    // Detect ON/OFF state change
    IF aUnits[i].bPresVal <> aPrevState[i] THEN
        // --------------------------------------------------------
        // (a) Send TwinCAT message as before
        // --------------------------------------------------------
        IF aUnits[i].bPresVal THEN
            sMsgText := CONCAT(stUnit.sUnitName, ' is Turned ON');
        ELSE
            sMsgText := CONCAT(stUnit.sUnitName, ' is Turned OFF');
        END_IF

        fbMsg.CreateEx(TC_EVENTS.UnitPowerStatus.EventPowerStatus, 0);
        fbMsg.ipArguments.AddString(sMsgText);
        fbMsg.Send(0);

        // --------------------------------------------------------
        // (b) Push event to global CSV queue (for P_CSVWrite_TextMode)
        // --------------------------------------------------------
        IF g_iCount < g_CSV_BUF_SIZE THEN
            g_aUnitName[g_iWriteIdx] := stUnit.sUnitName;
            g_aState[g_iWriteIdx]    := aUnits[i].bPresVal;
            g_iWriteIdx := g_iWriteIdx + 1;
            IF g_iWriteIdx > g_CSV_BUF_SIZE THEN g_iWriteIdx := 1; END_IF
            g_iCount := g_iCount + 1;
        END_IF

        // --------------------------------------------------------
        // (c) Update previous state
        // --------------------------------------------------------
        aPrevState[i] := aUnits[i].bPresVal;
    END_IF
END_FOR

// ------------------------------------------------------------
// Optional debug info
// ------------------------------------------------------------
sDebug := CONCAT('Queued=', INT_TO_STRING(g_iCount));

END_FUNCTION_BLOCK

// ---- POUs/FB_EventLogger/FB_EventFMZ2.TcPOU
FUNCTION_BLOCK FB_EventFMZ2
VAR_INPUT
	FB_Bacnet : FB_BACnet_DAIKIN_MasterStation_III_No_1;
END_VAR
VAR_OUTPUT
	sDebug : STRING(200);
END_VAR
VAR
	fbMsg : FB_TcMessage;
	aUnits : ARRAY[1..8] OF AC_Unit_Status;
	stUnit   : AC_Unit_Status;
	i: INT;
	sMsgText: STRING;

END_VAR
VAR RETAIN
	aPrevState : ARRAY[1..8] OF BOOL := [FALSE(*8*)];
END_VAR


aUnits[1].bPresVal := FB_Bacnet.StartStopStatus_096.bPresVal;
aUnits[1].sUnitName := 'FMZ-PC-1 (3-00)';
aUnits[2].bPresVal := FB_Bacnet.StartStopStatus_097.bPresVal;
aUnits[2].sUnitName := 'FMZ-PC-2 (3-01)';
aUnits[3].bPresVal := FB_Bacnet.StartStopStatus_098.bPresVal;
aUnits[3].sUnitName := 'FMZ-PC-3 (3-02)';
aUnits[4].bPresVal := FB_Bacnet.StartStopStatus_099.bPresVal;
aUnits[4].sUnitName := 'FMZ-PC-4 (3-03)';
aUnits[5].bPresVal := FB_Bacnet.StartStopStatus_100.bPresVal;
aUnits[5].sUnitName := 'FMZ-PC-5 (3-04)';
aUnits[6].bPresVal := FB_Bacnet.StartStopStatus_101.bPresVal;
aUnits[6].sUnitName := 'FMZ-PC-6 (3-05)';
aUnits[7].bPresVal := FB_Bacnet.StartStopStatus_102.bPresVal;
aUnits[7].sUnitName := 'FMZ-PC-7 (3-06)';
aUnits[8].bPresVal := FB_Bacnet.StartStopStatus_103.bPresVal;
aUnits[8].sUnitName := 'FMZ-PC-8 (3-07)';

FOR i := 1 TO 8 DO
    stUnit := aUnits[i];

    // Detect ON/OFF state change
    IF aUnits[i].bPresVal <> aPrevState[i] THEN
        // --------------------------------------------------------
        // (a) Send TwinCAT message as before
        // --------------------------------------------------------
        IF aUnits[i].bPresVal THEN
            sMsgText := CONCAT(stUnit.sUnitName, ' is Turned ON');
        ELSE
            sMsgText := CONCAT(stUnit.sUnitName, ' is Turned OFF');
        END_IF

        fbMsg.CreateEx(TC_EVENTS.UnitPowerStatus.EventPowerStatus, 0);
        fbMsg.ipArguments.AddString(sMsgText);
        fbMsg.Send(0);

        // --------------------------------------------------------
        // (b) Push event to global CSV queue (for P_CSVWrite_TextMode)
        // --------------------------------------------------------
        IF g_iCount < g_CSV_BUF_SIZE THEN
            g_aUnitName[g_iWriteIdx] := stUnit.sUnitName;
            g_aState[g_iWriteIdx]    := aUnits[i].bPresVal;
            g_iWriteIdx := g_iWriteIdx + 1;
            IF g_iWriteIdx > g_CSV_BUF_SIZE THEN g_iWriteIdx := 1; END_IF
            g_iCount := g_iCount + 1;
        END_IF

        // --------------------------------------------------------
        // (c) Update previous state
        // --------------------------------------------------------
        aPrevState[i] := aUnits[i].bPresVal;
    END_IF
END_FOR

// ------------------------------------------------------------
// Optional debug info
// ------------------------------------------------------------
sDebug := CONCAT('Queued=', INT_TO_STRING(g_iCount));

END_FUNCTION_BLOCK

// ---- POUs/FB_EventLogger/FB_EventF2.TcPOU
FUNCTION_BLOCK FB_EventF2
VAR_INPUT
	FB_Bacnet : FB_BACnet_DAIKIN_MasterStation_III_No_1;
END_VAR
VAR_OUTPUT
	sDebug : STRING(200);
END_VAR
VAR
	fbMsg : FB_TcMessage;
	aUnits : ARRAY[1..23] OF AC_Unit_Status;
	stUnit   : AC_Unit_Status;
	i: INT;
	sMsgText: STRING;
END_VAR
VAR RETAIN
	aPrevState : ARRAY[1..23] OF BOOL := [FALSE(*23*)];
END_VAR


aUnits[1].bPresVal := FB_Bacnet.StartStopStatus_128.bPresVal;
aUnits[1].sUnitName := 'F2-1 (1-00)';
aUnits[2].bPresVal := FB_Bacnet.StartStopStatus_129.bPresVal;
aUnits[2].sUnitName := 'F2-2 (1-01)';
aUnits[3].bPresVal := FB_Bacnet.StartStopStatus_130.bPresVal;
aUnits[3].sUnitName := 'F2-3 (1-02)';
aUnits[4].bPresVal := FB_Bacnet.StartStopStatus_131.bPresVal;
aUnits[4].sUnitName := 'F2-4 (1-03)';
aUnits[5].bPresVal := FB_Bacnet.StartStopStatus_132.bPresVal;
aUnits[5].sUnitName := 'F2-5 (1-04)';
aUnits[6].bPresVal := FB_Bacnet.StartStopStatus_133.bPresVal;
aUnits[6].sUnitName := 'F2-6 (1-05)';
aUnits[7].bPresVal := FB_Bacnet.StartStopStatus_134.bPresVal;
aUnits[7].sUnitName := 'F2-7 (1-06)';
aUnits[8].bPresVal := FB_Bacnet.StartStopStatus_135.bPresVal;
aUnits[8].sUnitName := 'F2-8 (1-07)';
aUnits[9].bPresVal := FB_Bacnet.StartStopStatus_136.bPresVal;
aUnits[9].sUnitName := 'F2-9 (1-08)';
aUnits[10].bPresVal := FB_Bacnet.StartStopStatus_137.bPresVal;
aUnits[10].sUnitName := 'F2-10 (1-09)';
aUnits[11].bPresVal := FB_Bacnet.StartStopStatus_138.bPresVal;
aUnits[11].sUnitName := 'F2-11 (1-10)';
aUnits[12].bPresVal := FB_Bacnet.StartStopStatus_139.bPresVal;
aUnits[12].sUnitName := 'F2-12 (1-11)';
//aUnits[13].bPresVal := FB_Bacnet.StartStopStatus_140.bPresVal;
//aUnits[13].sUnitName := 'F2-13 (1-12)';
aUnits[14].bPresVal := FB_Bacnet.StartStopStatus_141.bPresVal;
aUnits[14].sUnitName := 'F2-14 (1-13)';
aUnits[15].bPresVal := FB_Bacnet.StartStopStatus_142.bPresVal;
aUnits[15].sUnitName := 'F2-15 (1-14)';
aUnits[16].bPresVal := FB_Bacnet.StartStopStatus_143.bPresVal;
aUnits[16].sUnitName := 'F2-16 (1-15)';
aUnits[17].bPresVal := FB_Bacnet.StartStopStatus_144.bPresVal;
aUnits[17].sUnitName := 'F2-17 (2-00)';
aUnits[18].bPresVal := FB_Bacnet.StartStopStatus_145.bPresVal;
aUnits[18].sUnitName := 'F2-18 (2-01)';
aUnits[19].bPresVal := FB_Bacnet.StartStopStatus_146.bPresVal;
aUnits[19].sUnitName := 'F2-19 (2-02)';
aUnits[20].bPresVal := FB_Bacnet.StartStopStatus_147.bPresVal;
aUnits[20].sUnitName := 'F2-20 (2-03)';
aUnits[21].bPresVal := FB_Bacnet.StartStopStatus_148.bPresVal;
aUnits[21].sUnitName := 'F2-21 (2-04)';
aUnits[22].bPresVal := FB_Bacnet.StartStopStatus_176.bPresVal;
aUnits[22].sUnitName := 'F2-IT-1 (4-00)';
//aUnits[23].bPresVal := FB_Bacnet.StartStopStatus_177.bPresVal;
//aUnits[23].sUnitName := 'F2-IT-2 (4-01)';

FOR i := 1 TO 23 DO
    stUnit := aUnits[i];

    // Detect ON/OFF state change
    IF aUnits[i].bPresVal <> aPrevState[i] THEN
        // --------------------------------------------------------
        // (a) Send TwinCAT message as before
        // --------------------------------------------------------
        IF aUnits[i].bPresVal THEN
            sMsgText := CONCAT(stUnit.sUnitName, ' is Turned ON');
        ELSE
            sMsgText := CONCAT(stUnit.sUnitName, ' is Turned OFF');
        END_IF

        fbMsg.CreateEx(TC_EVENTS.UnitPowerStatus.EventPowerStatus, 0);
        fbMsg.ipArguments.AddString(sMsgText);
        fbMsg.Send(0);

        // --------------------------------------------------------
        // (b) Push event to global CSV queue (for P_CSVWrite_TextMode)
        // --------------------------------------------------------
        IF g_iCount < g_CSV_BUF_SIZE THEN
            g_aUnitName[g_iWriteIdx] := stUnit.sUnitName;
            g_aState[g_iWriteIdx]    := aUnits[i].bPresVal;
            g_iWriteIdx := g_iWriteIdx + 1;
            IF g_iWriteIdx > g_CSV_BUF_SIZE THEN g_iWriteIdx := 1; END_IF
            g_iCount := g_iCount + 1;
        END_IF

        // --------------------------------------------------------
        // (c) Update previous state
        // --------------------------------------------------------
        aPrevState[i] := aUnits[i].bPresVal;
    END_IF
END_FOR

// ------------------------------------------------------------
// Optional debug info
// ------------------------------------------------------------
sDebug := CONCAT('Queued=', INT_TO_STRING(g_iCount));

END_FUNCTION_BLOCK

// ---- POUs/FB_EventLogger/FB_EventF3.TcPOU
FUNCTION_BLOCK FB_EventF3
VAR_INPUT
	FB_Bacnet : FB_BACnet_DAIKIN_MasterStation_III_No_1;
END_VAR
VAR_OUTPUT
	sDebug : STRING(200);
END_VAR
VAR
	fbMsg : FB_TcMessage;
	aUnits : ARRAY[1..22] OF AC_Unit_Status;
	stUnit   : AC_Unit_Status;
	i: INT;
	sMsgText: STRING;

END_VAR
VAR RETAIN
	aPrevState : ARRAY[1..22] OF BOOL := [FALSE(*22*)];
END_VAR


//aUnits[1].bPresVal := FB_Bacnet.StartStopStatus_192.bPresVal;
//aUnits[1].sUnitName := 'F3-1 (1-00)';
aUnits[2].bPresVal := FB_Bacnet.StartStopStatus_193.bPresVal;
aUnits[2].sUnitName := 'F3-2 (1-01)';
aUnits[3].bPresVal := FB_Bacnet.StartStopStatus_194.bPresVal;
aUnits[3].sUnitName := 'F3-3 (1-02)';
aUnits[4].bPresVal := FB_Bacnet.StartStopStatus_195.bPresVal;
aUnits[4].sUnitName := 'F3-4 (1-03)';
aUnits[5].bPresVal := FB_Bacnet.StartStopStatus_196.bPresVal;
aUnits[5].sUnitName := 'F3-5 (1-04)';
aUnits[6].bPresVal := FB_Bacnet.StartStopStatus_197.bPresVal;
aUnits[6].sUnitName := 'F3-6 (1-05)';
aUnits[7].bPresVal := FB_Bacnet.StartStopStatus_198.bPresVal;
aUnits[7].sUnitName := 'F3-7 (1-06)';
aUnits[8].bPresVal := FB_Bacnet.StartStopStatus_199.bPresVal;
aUnits[8].sUnitName := 'F3-8 (1-07)';
aUnits[9].bPresVal := FB_Bacnet.StartStopStatus_200.bPresVal;
aUnits[9].sUnitName := 'F3-9 (1-08)';
aUnits[10].bPresVal := FB_Bacnet.StartStopStatus_201.bPresVal;
aUnits[10].sUnitName := 'F3-10 (1-09)';
aUnits[11].bPresVal := FB_Bacnet.StartStopStatus_202.bPresVal;
aUnits[11].sUnitName := 'F3-11 (1-10)';
aUnits[12].bPresVal := FB_Bacnet.StartStopStatus_203.bPresVal;
aUnits[12].sUnitName := 'F3-12 (1-11)';
aUnits[13].bPresVal := FB_Bacnet.StartStopStatus_204.bPresVal;
aUnits[13].sUnitName := 'F3-13 (1-12)';
aUnits[14].bPresVal := FB_Bacnet.StartStopStatus_205.bPresVal;
aUnits[14].sUnitName := 'F3-14 (1-13)';
aUnits[15].bPresVal := FB_Bacnet.StartStopStatus_206.bPresVal;
aUnits[15].sUnitName := 'F3-15 (1-14)';
aUnits[16].bPresVal := FB_Bacnet.StartStopStatus_207.bPresVal;
aUnits[16].sUnitName := 'F3-16 (1-15)';
aUnits[17].bPresVal := FB_Bacnet.StartStopStatus_208.bPresVal;
aUnits[17].sUnitName := 'F3-17 (2-00)';
aUnits[18].bPresVal := FB_Bacnet.StartStopStatus_209.bPresVal;
aUnits[18].sUnitName := 'F3-18 (2-01)';
aUnits[19].bPresVal := FB_Bacnet.StartStopStatus_210.bPresVal;
aUnits[19].sUnitName := 'F3-19 (2-02)';
aUnits[20].bPresVal := FB_Bacnet.StartStopStatus_211.bPresVal;
aUnits[20].sUnitName := 'F3-20 (2-03)';
aUnits[21].bPresVal := FB_Bacnet.StartStopStatus_212.bPresVal;
aUnits[21].sUnitName := 'F3-21 (2-04)';
aUnits[22].bPresVal := FB_Bacnet.StartStopStatus_224.bPresVal;
aUnits[22].sUnitName := 'F3-Lobi (3-00)';

FOR i := 1 TO 22 DO
    stUnit := aUnits[i];

    // Detect ON/OFF state change
    IF aUnits[i].bPresVal <> aPrevState[i] THEN
        // --------------------------------------------------------
        // (a) Send TwinCAT message as before
        // --------------------------------------------------------
        IF aUnits[i].bPresVal THEN
            sMsgText := CONCAT(stUnit.sUnitName, ' is Turned ON');
        ELSE
            sMsgText := CONCAT(stUnit.sUnitName, ' is Turned OFF');
        END_IF

        fbMsg.CreateEx(TC_EVENTS.UnitPowerStatus.EventPowerStatus, 0);
        fbMsg.ipArguments.AddString(sMsgText);
        fbMsg.Send(0);

        // --------------------------------------------------------
        // (b) Push event to global CSV queue (for P_CSVWrite_TextMode)
        // --------------------------------------------------------
        IF g_iCount < g_CSV_BUF_SIZE THEN
            g_aUnitName[g_iWriteIdx] := stUnit.sUnitName;
            g_aState[g_iWriteIdx]    := aUnits[i].bPresVal;
            g_iWriteIdx := g_iWriteIdx + 1;
            IF g_iWriteIdx > g_CSV_BUF_SIZE THEN g_iWriteIdx := 1; END_IF
            g_iCount := g_iCount + 1;
        END_IF

        // --------------------------------------------------------
        // (c) Update previous state
        // --------------------------------------------------------
        aPrevState[i] := aUnits[i].bPresVal;
    END_IF
END_FOR

// ------------------------------------------------------------
// Optional debug info
// ------------------------------------------------------------
sDebug := CONCAT('Queued=', INT_TO_STRING(g_iCount));

END_FUNCTION_BLOCK

// ---- POUs/FB_EventLogger/FB_EventF5.TcPOU
FUNCTION_BLOCK FB_EventF5
VAR_INPUT
	FB_Bacnet : FB_BACnet_DAIKIN_MasterStation_III_No_2;
    FB_Bacnet_b : FB_BACnet_DAIKIN_MasterStation_III_No_1;
END_VAR
VAR_OUTPUT
	sDebug : STRING(200);
END_VAR
VAR
	fbMsg : FB_TcMessage;
	aUnits : ARRAY[1..22] OF AC_Unit_Status;
	stUnit   : AC_Unit_Status;
	i: INT;
	sMsgText: STRING;

END_VAR
VAR RETAIN
	aPrevState : ARRAY[1..22] OF BOOL := [FALSE(*22*)];
END_VAR


aUnits[1].bPresVal := FB_Bacnet.StartStopStatus_000.bPresVal;
aUnits[1].sUnitName := 'F5-A1 (1-00)';
aUnits[2].bPresVal := FB_Bacnet.StartStopStatus_001.bPresVal;
aUnits[2].sUnitName := 'F5-A2 (1-01)';
aUnits[3].bPresVal := FB_Bacnet.StartStopStatus_002.bPresVal;
aUnits[3].sUnitName := 'F5-A3 (1-02)';
aUnits[4].bPresVal := FB_Bacnet.StartStopStatus_003.bPresVal;
aUnits[4].sUnitName := 'F5-A4 (1-03)';
aUnits[5].bPresVal := FB_Bacnet.StartStopStatus_004.bPresVal;
aUnits[5].sUnitName := 'F5-B1 (1-04)';
aUnits[6].bPresVal := FB_Bacnet.StartStopStatus_005.bPresVal;
aUnits[6].sUnitName := 'F5-B2 (1-05)';
aUnits[7].bPresVal := FB_Bacnet.StartStopStatus_006.bPresVal;
aUnits[7].sUnitName := 'F5-C1 (1-06)';
aUnits[8].bPresVal := FB_Bacnet.StartStopStatus_007.bPresVal;
aUnits[8].sUnitName := 'F5-C2 (1-07)';
aUnits[9].bPresVal := FB_Bacnet.StartStopStatus_008.bPresVal;
aUnits[9].sUnitName := 'F5-D1 (1-08)';
aUnits[10].bPresVal := FB_Bacnet.StartStopStatus_009.bPresVal;
aUnits[10].sUnitName := 'F5-D2 (1-09)';
aUnits[11].bPresVal := FB_Bacnet.StartStopStatus_010.bPresVal;
aUnits[11].sUnitName := 'F5-D3 (1-10)';
aUnits[12].bPresVal := FB_Bacnet.StartStopStatus_011.bPresVal;
aUnits[12].sUnitName := 'F5-D4 (1-11)';
aUnits[13].bPresVal := FB_Bacnet.StartStopStatus_012.bPresVal;
aUnits[13].sUnitName := 'F5-D5 (1-12)';
aUnits[14].bPresVal := FB_Bacnet.StartStopStatus_013.bPresVal;
aUnits[14].sUnitName := 'F5-D6 (1-13)';
aUnits[15].bPresVal := FB_Bacnet.StartStopStatus_014.bPresVal;
aUnits[15].sUnitName := 'F5-E1 (1-14)';
aUnits[16].bPresVal := FB_Bacnet.StartStopStatus_015.bPresVal;
aUnits[16].sUnitName := 'F5-E2 (1-15)';
aUnits[17].bPresVal := FB_Bacnet.StartStopStatus_016.bPresVal;
aUnits[17].sUnitName := 'F5-F1 (2-00)';
aUnits[18].bPresVal := FB_Bacnet.StartStopStatus_017.bPresVal;
aUnits[18].sUnitName := 'F5-F2 (2-01)';
aUnits[19].bPresVal := FB_Bacnet.StartStopStatus_018.bPresVal;
aUnits[19].sUnitName := 'F5-G1 (2-02)';
aUnits[20].bPresVal := FB_Bacnet.StartStopStatus_019.bPresVal;
aUnits[20].sUnitName := 'F5-G2 (2-03)';
aUnits[21].bPresVal := FB_Bacnet.StartStopStatus_020.bPresVal;
aUnits[21].sUnitName := 'F5-G3 (2-04)';
aUnits[22].bPresVal := FB_Bacnet_b.StartStopStatus_225.bPresVal;
aUnits[22].sUnitName := 'F5-Lobi (3-01)';

FOR i := 1 TO 22 DO
    stUnit := aUnits[i];

    // Detect ON/OFF state change
    IF aUnits[i].bPresVal <> aPrevState[i] THEN
        // --------------------------------------------------------
        // (a) Send TwinCAT message as before
        // --------------------------------------------------------
        IF aUnits[i].bPresVal THEN
            sMsgText := CONCAT(stUnit.sUnitName, ' is Turned ON');
        ELSE
            sMsgText := CONCAT(stUnit.sUnitName, ' is Turned OFF');
        END_IF

        fbMsg.CreateEx(TC_EVENTS.UnitPowerStatus.EventPowerStatus, 0);
        fbMsg.ipArguments.AddString(sMsgText);
        fbMsg.Send(0);

        // --------------------------------------------------------
        // (b) Push event to global CSV queue (for P_CSVWrite_TextMode)
        // --------------------------------------------------------
        IF g_iCount < g_CSV_BUF_SIZE THEN
            g_aUnitName[g_iWriteIdx] := stUnit.sUnitName;
            g_aState[g_iWriteIdx]    := aUnits[i].bPresVal;
            g_iWriteIdx := g_iWriteIdx + 1;
            IF g_iWriteIdx > g_CSV_BUF_SIZE THEN g_iWriteIdx := 1; END_IF
            g_iCount := g_iCount + 1;
        END_IF

        // --------------------------------------------------------
        // (c) Update previous state
        // --------------------------------------------------------
        aPrevState[i] := aUnits[i].bPresVal;
    END_IF
END_FOR

// ------------------------------------------------------------
// Optional debug info
// ------------------------------------------------------------
sDebug := CONCAT('Queued=', INT_TO_STRING(g_iCount));

END_FUNCTION_BLOCK

// ---- POUs/FB_EventLogger/FB_EventF6.TcPOU
FUNCTION_BLOCK FB_EventF6
VAR_INPUT
	FB_Bacnet : FB_BACnet_DAIKIN_MasterStation_III_No_2;
    FB_Bacnet_b : FB_BACnet_DAIKIN_MasterStation_III_No_1;
END_VAR
VAR_OUTPUT
	sDebug : STRING(200);
END_VAR
VAR
	fbMsg : FB_TcMessage;
	aUnits : ARRAY[1..22] OF AC_Unit_Status;
	stUnit   : AC_Unit_Status;
	i: INT;
	sMsgText: STRING;

END_VAR
VAR RETAIN
	aPrevState : ARRAY[1..22] OF BOOL := [FALSE(*22*)];
END_VAR


aUnits[1].bPresVal := FB_Bacnet.StartStopStatus_064.bPresVal;
aUnits[1].sUnitName := 'F6-A1 (1-00)';
aUnits[2].bPresVal := FB_Bacnet.StartStopStatus_065.bPresVal;
aUnits[2].sUnitName := 'F6-A2 (1-01)';
aUnits[3].bPresVal := FB_Bacnet.StartStopStatus_066.bPresVal;
aUnits[3].sUnitName := 'F6-A3 (1-02)';
aUnits[4].bPresVal := FB_Bacnet.StartStopStatus_067.bPresVal;
aUnits[4].sUnitName := 'F6-A4 (1-03)';
aUnits[5].bPresVal := FB_Bacnet.StartStopStatus_068.bPresVal;
aUnits[5].sUnitName := 'F6-B1 (1-04)';
aUnits[6].bPresVal := FB_Bacnet.StartStopStatus_069.bPresVal;
aUnits[6].sUnitName := 'F6-B2 (1-05)';
aUnits[7].bPresVal := FB_Bacnet.StartStopStatus_070.bPresVal;
aUnits[7].sUnitName := 'F6-C1 (1-06)';
aUnits[8].bPresVal := FB_Bacnet.StartStopStatus_071.bPresVal;
aUnits[8].sUnitName := 'F6-C2 (1-07)';
aUnits[9].bPresVal := FB_Bacnet.StartStopStatus_072.bPresVal;
aUnits[9].sUnitName := 'F6-D1 (1-08)';
aUnits[10].bPresVal := FB_Bacnet.StartStopStatus_073.bPresVal;
aUnits[10].sUnitName := 'F6-D2 (1-09)';
aUnits[11].bPresVal := FB_Bacnet.StartStopStatus_074.bPresVal;
aUnits[11].sUnitName := 'F6-D3 (1-10)';
aUnits[12].bPresVal := FB_Bacnet.StartStopStatus_075.bPresVal;
aUnits[12].sUnitName := 'F6-D4 (1-11)';
aUnits[13].bPresVal := FB_Bacnet.StartStopStatus_076.bPresVal;
aUnits[13].sUnitName := 'F6-D5 (1-12)';
aUnits[14].bPresVal := FB_Bacnet.StartStopStatus_077.bPresVal;
aUnits[14].sUnitName := 'F6-D6 (1-13)';
aUnits[15].bPresVal := FB_Bacnet.StartStopStatus_078.bPresVal;
aUnits[15].sUnitName := 'F6-E1 (1-14)';
aUnits[16].bPresVal := FB_Bacnet.StartStopStatus_079.bPresVal;
aUnits[16].sUnitName := 'F6-E2 (1-15)';
aUnits[17].bPresVal := FB_Bacnet.StartStopStatus_080.bPresVal;
aUnits[17].sUnitName := 'F6-F1 (2-00)';
aUnits[18].bPresVal := FB_Bacnet.StartStopStatus_081.bPresVal;
aUnits[18].sUnitName := 'F6-F2 (2-01)';
aUnits[19].bPresVal := FB_Bacnet.StartStopStatus_082.bPresVal;
aUnits[19].sUnitName := 'F6-G1 (2-02)';
aUnits[20].bPresVal := FB_Bacnet.StartStopStatus_083.bPresVal;
aUnits[20].sUnitName := 'F6-G2 (2-03)';
aUnits[21].bPresVal := FB_Bacnet.StartStopStatus_084.bPresVal;
aUnits[21].sUnitName := 'F6-G3 (2-04)';
aUnits[22].bPresVal := FB_Bacnet_b.StartStopStatus_226.bPresVal;
aUnits[22].sUnitName := 'F6-Lobi (3-02)';

FOR i := 1 TO 22 DO
    stUnit := aUnits[i];

    // Detect ON/OFF state change
    IF aUnits[i].bPresVal <> aPrevState[i] THEN
        // --------------------------------------------------------
        // (a) Send TwinCAT message as before
        // --------------------------------------------------------
        IF aUnits[i].bPresVal THEN
            sMsgText := CONCAT(stUnit.sUnitName, ' is Turned ON');
        ELSE
            sMsgText := CONCAT(stUnit.sUnitName, ' is Turned OFF');
        END_IF

        fbMsg.CreateEx(TC_EVENTS.UnitPowerStatus.EventPowerStatus, 0);
        fbMsg.ipArguments.AddString(sMsgText);
        fbMsg.Send(0);

        // --------------------------------------------------------
        // (b) Push event to global CSV queue (for P_CSVWrite_TextMode)
        // --------------------------------------------------------
        IF g_iCount < g_CSV_BUF_SIZE THEN
            g_aUnitName[g_iWriteIdx] := stUnit.sUnitName;
            g_aState[g_iWriteIdx]    := aUnits[i].bPresVal;
            g_iWriteIdx := g_iWriteIdx + 1;
            IF g_iWriteIdx > g_CSV_BUF_SIZE THEN g_iWriteIdx := 1; END_IF
            g_iCount := g_iCount + 1;
        END_IF

        // --------------------------------------------------------
        // (c) Update previous state
        // --------------------------------------------------------
        aPrevState[i] := aUnits[i].bPresVal;
    END_IF
END_FOR

// ------------------------------------------------------------
// Optional debug info
// ------------------------------------------------------------
sDebug := CONCAT('Queued=', INT_TO_STRING(g_iCount));

END_FUNCTION_BLOCK

// ---- POUs/FB_EventLogger/FB_EventF7.TcPOU
FUNCTION_BLOCK FB_EventF7
VAR_INPUT
	FB_Bacnet : FB_BACnet_DAIKIN_MasterStation_III_No_2;
    FB_Bacnet_b : FB_BACnet_DAIKIN_MasterStation_III_No_1;
END_VAR
VAR_OUTPUT
	sDebug : STRING(200);
END_VAR
VAR
	fbMsg : FB_TcMessage;
	aUnits : ARRAY[1..24] OF AC_Unit_Status;
	stUnit   : AC_Unit_Status;
	i: INT;
	sMsgText: STRING;

END_VAR
VAR RETAIN
	aPrevState : ARRAY[1..24] OF BOOL := [FALSE(*24*)];
END_VAR


aUnits[1].bPresVal := FB_Bacnet.StartStopStatus_128.bPresVal;
aUnits[1].sUnitName := 'F7-A1 (1-00)';
aUnits[2].bPresVal := FB_Bacnet.StartStopStatus_129.bPresVal;
aUnits[2].sUnitName := 'F7-A2 (1-01)';
aUnits[3].bPresVal := FB_Bacnet.StartStopStatus_130.bPresVal;
aUnits[3].sUnitName := 'F7-A3 (1-02)';
aUnits[4].bPresVal := FB_Bacnet.StartStopStatus_131.bPresVal;
aUnits[4].sUnitName := 'F7-A4 (1-03)';
aUnits[5].bPresVal := FB_Bacnet.StartStopStatus_132.bPresVal;
aUnits[5].sUnitName := 'F7-B1 (1-04)';
aUnits[6].bPresVal := FB_Bacnet.StartStopStatus_133.bPresVal;
aUnits[6].sUnitName := 'F7-B2 (1-05)';
aUnits[7].bPresVal := FB_Bacnet.StartStopStatus_134.bPresVal;
aUnits[7].sUnitName := 'F7-C1 (1-06)';
aUnits[8].bPresVal := FB_Bacnet.StartStopStatus_135.bPresVal;
aUnits[8].sUnitName := 'F7-C2 (1-07)';
aUnits[9].bPresVal := FB_Bacnet.StartStopStatus_136.bPresVal;
aUnits[9].sUnitName := 'F7-D1 (1-08)';
aUnits[10].bPresVal := FB_Bacnet.StartStopStatus_137.bPresVal;
aUnits[10].sUnitName := 'F7-D2 (1-09)';
aUnits[11].bPresVal := FB_Bacnet.StartStopStatus_138.bPresVal;
aUnits[11].sUnitName := 'F7-D3 (1-10)';
aUnits[12].bPresVal := FB_Bacnet.StartStopStatus_139.bPresVal;
aUnits[12].sUnitName := 'F7-D4 (1-11)';
aUnits[13].bPresVal := FB_Bacnet.StartStopStatus_140.bPresVal;
aUnits[13].sUnitName := 'F7-D5 (1-12)';
aUnits[14].bPresVal := FB_Bacnet.StartStopStatus_141.bPresVal;
aUnits[14].sUnitName := 'F7-D6 (1-13)';
aUnits[15].bPresVal := FB_Bacnet.StartStopStatus_142.bPresVal;
aUnits[15].sUnitName := 'F7-E1 (1-14)';
aUnits[16].bPresVal := FB_Bacnet.StartStopStatus_143.bPresVal;
aUnits[16].sUnitName := 'F7-E2 (1-15)';
aUnits[17].bPresVal := FB_Bacnet.StartStopStatus_144.bPresVal;
aUnits[17].sUnitName := 'F7-F1 (2-00)';
aUnits[18].bPresVal := FB_Bacnet.StartStopStatus_145.bPresVal;
aUnits[18].sUnitName := 'F7-F2 (2-01)';
aUnits[19].bPresVal := FB_Bacnet.StartStopStatus_146.bPresVal;
aUnits[19].sUnitName := 'F7-G1 (2-02)';
aUnits[20].bPresVal := FB_Bacnet.StartStopStatus_147.bPresVal;
aUnits[20].sUnitName := 'F7-G2 (2-03)';
aUnits[21].bPresVal := FB_Bacnet.StartStopStatus_148.bPresVal;
aUnits[21].sUnitName := 'F7-G3 (2-04)';
aUnits[22].bPresVal := FB_Bacnet.StartStopStatus_176.bPresVal;
aUnits[22].sUnitName := 'F7-IT-1 (4-00)';
aUnits[23].bPresVal := FB_Bacnet_b.StartStopStatus_241.bPresVal;
aUnits[23].sUnitName := 'F7-IT-2 (4-01)';
aUnits[24].bPresVal := FB_Bacnet_b.StartStopStatus_227.bPresVal;
aUnits[24].sUnitName := 'F7-Lobi (3-03)';

FOR i := 1 TO 24 DO
    stUnit := aUnits[i];

    // Detect ON/OFF state change
    IF aUnits[i].bPresVal <> aPrevState[i] THEN
        // --------------------------------------------------------
        // (a) Send TwinCAT message as before
        // --------------------------------------------------------
        IF aUnits[i].bPresVal THEN
            sMsgText := CONCAT(stUnit.sUnitName, ' is Turned ON');
        ELSE
            sMsgText := CONCAT(stUnit.sUnitName, ' is Turned OFF');
        END_IF

        fbMsg.CreateEx(TC_EVENTS.UnitPowerStatus.EventPowerStatus, 0);
        fbMsg.ipArguments.AddString(sMsgText);
        fbMsg.Send(0);

        // --------------------------------------------------------
        // (b) Push event to global CSV queue (for P_CSVWrite_TextMode)
        // --------------------------------------------------------
        IF g_iCount < g_CSV_BUF_SIZE THEN
            g_aUnitName[g_iWriteIdx] := stUnit.sUnitName;
            g_aState[g_iWriteIdx]    := aUnits[i].bPresVal;
            g_iWriteIdx := g_iWriteIdx + 1;
            IF g_iWriteIdx > g_CSV_BUF_SIZE THEN g_iWriteIdx := 1; END_IF
            g_iCount := g_iCount + 1;
        END_IF

        // --------------------------------------------------------
        // (c) Update previous state
        // --------------------------------------------------------
        aPrevState[i] := aUnits[i].bPresVal;
    END_IF
END_FOR

// ------------------------------------------------------------
// Optional debug info
// ------------------------------------------------------------
sDebug := CONCAT('Queued=', INT_TO_STRING(g_iCount));

END_FUNCTION_BLOCK

// ---- POUs/FB_EventLogger/FB_EventF8.TcPOU
FUNCTION_BLOCK FB_EventF8
VAR_INPUT
	FB_Bacnet : FB_BACnet_DAIKIN_MasterStation_III_No_2;
END_VAR
VAR_OUTPUT
	sDebug : STRING(200);
END_VAR
VAR
	fbMsg : FB_TcMessage;
	aUnits : ARRAY[1..22] OF AC_Unit_Status;
	stUnit   : AC_Unit_Status;
	i: INT;
	sMsgText: STRING;

END_VAR
VAR RETAIN
	aPrevState : ARRAY[1..22] OF BOOL := [FALSE(*22*)];
END_VAR


aUnits[1].bPresVal := FB_Bacnet.StartStopStatus_192.bPresVal;
aUnits[1].sUnitName := 'F8-A1 (1-00)';
aUnits[2].bPresVal := FB_Bacnet.StartStopStatus_193.bPresVal;
aUnits[2].sUnitName := 'F8-A2 (1-01)';
aUnits[3].bPresVal := FB_Bacnet.StartStopStatus_194.bPresVal;
aUnits[3].sUnitName := 'F8-A3 (1-02)';
aUnits[4].bPresVal := FB_Bacnet.StartStopStatus_195.bPresVal;
aUnits[4].sUnitName := 'F8-A4 (1-03)';
aUnits[5].bPresVal := FB_Bacnet.StartStopStatus_196.bPresVal;
aUnits[5].sUnitName := 'F8-B1 (1-04)';
aUnits[6].bPresVal := FB_Bacnet.StartStopStatus_197.bPresVal;
aUnits[6].sUnitName := 'F8-B2 (1-05)';
aUnits[7].bPresVal := FB_Bacnet.StartStopStatus_198.bPresVal;
aUnits[7].sUnitName := 'F8-C1 (1-06)';
aUnits[8].bPresVal := FB_Bacnet.StartStopStatus_199.bPresVal;
aUnits[8].sUnitName := 'F8-C2 (1-07)';
aUnits[9].bPresVal := FB_Bacnet.StartStopStatus_200.bPresVal;
aUnits[9].sUnitName := 'F8-D1 (1-08)';
aUnits[10].bPresVal := FB_Bacnet.StartStopStatus_201.bPresVal;
aUnits[10].sUnitName := 'F8-D2 (1-09)';
aUnits[11].bPresVal := FB_Bacnet.StartStopStatus_202.bPresVal;
aUnits[11].sUnitName := 'F8-D3 (1-10)';
aUnits[12].bPresVal := FB_Bacnet.StartStopStatus_203.bPresVal;
aUnits[12].sUnitName := 'F8-D4 (1-11)';
aUnits[13].bPresVal := FB_Bacnet.StartStopStatus_204.bPresVal;
aUnits[13].sUnitName := 'F8-D5 (1-12)';
aUnits[14].bPresVal := FB_Bacnet.StartStopStatus_205.bPresVal;
aUnits[14].sUnitName := 'F8-D6 (1-13)';
aUnits[15].bPresVal := FB_Bacnet.StartStopStatus_206.bPresVal;
aUnits[15].sUnitName := 'F8-E1 (1-14)';
aUnits[16].bPresVal := FB_Bacnet.StartStopStatus_207.bPresVal;
aUnits[16].sUnitName := 'F8-E2 (1-15)';
aUnits[17].bPresVal := FB_Bacnet.StartStopStatus_208.bPresVal;
aUnits[17].sUnitName := 'F8-F1 (2-00)';
aUnits[18].bPresVal := FB_Bacnet.StartStopStatus_209.bPresVal;
aUnits[18].sUnitName := 'F8-F2 (2-01)';
aUnits[19].bPresVal := FB_Bacnet.StartStopStatus_210.bPresVal;
aUnits[19].sUnitName := 'F8-G1 (2-02)';
aUnits[20].bPresVal := FB_Bacnet.StartStopStatus_211.bPresVal;
aUnits[20].sUnitName := 'F8-G2 (2-03)';
aUnits[21].bPresVal := FB_Bacnet.StartStopStatus_212.bPresVal;
aUnits[21].sUnitName := 'F8-G3 (2-04)';
aUnits[22].bPresVal := FB_Bacnet.StartStopStatus_224.bPresVal;
aUnits[22].sUnitName := 'F8-Lobi (3-00)';


FOR i := 1 TO 22 DO
    stUnit := aUnits[i];

    // Detect ON/OFF state change
    IF aUnits[i].bPresVal <> aPrevState[i] THEN
        // --------------------------------------------------------
        // (a) Send TwinCAT message as before
        // --------------------------------------------------------
        IF aUnits[i].bPresVal THEN
            sMsgText := CONCAT(stUnit.sUnitName, ' is Turned ON');
        ELSE
            sMsgText := CONCAT(stUnit.sUnitName, ' is Turned OFF');
        END_IF

        fbMsg.CreateEx(TC_EVENTS.UnitPowerStatus.EventPowerStatus, 0);
        fbMsg.ipArguments.AddString(sMsgText);
        fbMsg.Send(0);

        // --------------------------------------------------------
        // (b) Push event to global CSV queue (for P_CSVWrite_TextMode)
        // --------------------------------------------------------
        IF g_iCount < g_CSV_BUF_SIZE THEN
            g_aUnitName[g_iWriteIdx] := stUnit.sUnitName;
            g_aState[g_iWriteIdx]    := aUnits[i].bPresVal;
            g_iWriteIdx := g_iWriteIdx + 1;
            IF g_iWriteIdx > g_CSV_BUF_SIZE THEN g_iWriteIdx := 1; END_IF
            g_iCount := g_iCount + 1;
        END_IF

        // --------------------------------------------------------
        // (c) Update previous state
        // --------------------------------------------------------
        aPrevState[i] := aUnits[i].bPresVal;
    END_IF
END_FOR

// ------------------------------------------------------------
// Optional debug info
// ------------------------------------------------------------
sDebug := CONCAT('Queued=', INT_TO_STRING(g_iCount));

END_FUNCTION_BLOCK

// ---- POUs/FB_EventLogger/FB_EventF9.TcPOU
FUNCTION_BLOCK FB_EventF9
VAR_INPUT
	FB_Bacnet : FB_BACnet_DAIKIN_MasterStation_III_No_3;
  FB_Bacnet_b : FB_BACnet_DAIKIN_MasterStation_III_No_2;
END_VAR
VAR_OUTPUT
	sDebug : STRING(200);
END_VAR
VAR
	fbMsg : FB_TcMessage;
	aUnits : ARRAY[1..22] OF AC_Unit_Status;
	stUnit   : AC_Unit_Status;
	i: INT;
	sMsgText: STRING;

END_VAR
VAR RETAIN
	aPrevState : ARRAY[1..22] OF BOOL := [FALSE(*22*)];
END_VAR


aUnits[1].bPresVal := FB_Bacnet.StartStopStatus_000.bPresVal;
aUnits[1].sUnitName := 'F9-A1 (1-00)';
aUnits[2].bPresVal := FB_Bacnet.StartStopStatus_001.bPresVal;
aUnits[2].sUnitName := 'F9-A2 (1-01)';
aUnits[3].bPresVal := FB_Bacnet.StartStopStatus_002.bPresVal;
aUnits[3].sUnitName := 'F9-A3 (1-02)';
aUnits[4].bPresVal := FB_Bacnet.StartStopStatus_003.bPresVal;
aUnits[4].sUnitName := 'F9-A4 (1-03)';
aUnits[5].bPresVal := FB_Bacnet.StartStopStatus_004.bPresVal;
aUnits[5].sUnitName := 'F9-B1 (1-04)';
aUnits[6].bPresVal := FB_Bacnet.StartStopStatus_005.bPresVal;
aUnits[6].sUnitName := 'F9-B2 (1-05)';
aUnits[7].bPresVal := FB_Bacnet.StartStopStatus_006.bPresVal;
aUnits[7].sUnitName := 'F9-C1 (1-06)';
aUnits[8].bPresVal := FB_Bacnet.StartStopStatus_007.bPresVal;
aUnits[8].sUnitName := 'F9-C2 (1-07)';
aUnits[9].bPresVal := FB_Bacnet.StartStopStatus_008.bPresVal;
aUnits[9].sUnitName := 'F9-D1 (1-08)';
aUnits[10].bPresVal := FB_Bacnet.StartStopStatus_009.bPresVal;
aUnits[10].sUnitName := 'F9-D2 (1-09)';
aUnits[11].bPresVal := FB_Bacnet.StartStopStatus_010.bPresVal;
aUnits[11].sUnitName := 'F9-D3 (1-10)';
aUnits[12].bPresVal := FB_Bacnet.StartStopStatus_011.bPresVal;
aUnits[12].sUnitName := 'F9-D4 (1-11)';
aUnits[13].bPresVal := FB_Bacnet.StartStopStatus_012.bPresVal;
aUnits[13].sUnitName := 'F9-D5 (1-12)';
aUnits[14].bPresVal := FB_Bacnet.StartStopStatus_013.bPresVal;
aUnits[14].sUnitName := 'F9-D6 (1-13)';
aUnits[15].bPresVal := FB_Bacnet.StartStopStatus_014.bPresVal;
aUnits[15].sUnitName := 'F9-E1 (1-14)';
aUnits[16].bPresVal := FB_Bacnet.StartStopStatus_015.bPresVal;
aUnits[16].sUnitName := 'F9-E2 (1-15)';
aUnits[17].bPresVal := FB_Bacnet.StartStopStatus_016.bPresVal;
aUnits[17].sUnitName := 'F9-F1 (2-00)';
aUnits[18].bPresVal := FB_Bacnet.StartStopStatus_017.bPresVal;
aUnits[18].sUnitName := 'F9-F2 (2-01)';
aUnits[19].bPresVal := FB_Bacnet.StartStopStatus_018.bPresVal;
aUnits[19].sUnitName := 'F9-G1 (2-02)';
aUnits[20].bPresVal := FB_Bacnet.StartStopStatus_019.bPresVal;
aUnits[20].sUnitName := 'F9-G2 (2-03)';
aUnits[21].bPresVal := FB_Bacnet.StartStopStatus_020.bPresVal;
aUnits[21].sUnitName := 'F9-G3 (2-04)';
aUnits[22].bPresVal := FB_Bacnet.StartStopStatus_225.bPresVal;
aUnits[22].sUnitName := 'F9-Lobi (3-01)';


FOR i := 1 TO 22 DO
    stUnit := aUnits[i];

    // Detect ON/OFF state change
    IF aUnits[i].bPresVal <> aPrevState[i] THEN
        // --------------------------------------------------------
        // (a) Send TwinCAT message as before
        // --------------------------------------------------------
        IF aUnits[i].bPresVal THEN
            sMsgText := CONCAT(stUnit.sUnitName, ' is Turned ON');
        ELSE
            sMsgText := CONCAT(stUnit.sUnitName, ' is Turned OFF');
        END_IF

        fbMsg.CreateEx(TC_EVENTS.UnitPowerStatus.EventPowerStatus, 0);
        fbMsg.ipArguments.AddString(sMsgText);
        fbMsg.Send(0);

        // --------------------------------------------------------
        // (b) Push event to global CSV queue (for P_CSVWrite_TextMode)
        // --------------------------------------------------------
        IF g_iCount < g_CSV_BUF_SIZE THEN
            g_aUnitName[g_iWriteIdx] := stUnit.sUnitName;
            g_aState[g_iWriteIdx]    := aUnits[i].bPresVal;
            g_iWriteIdx := g_iWriteIdx + 1;
            IF g_iWriteIdx > g_CSV_BUF_SIZE THEN g_iWriteIdx := 1; END_IF
            g_iCount := g_iCount + 1;
        END_IF

        // --------------------------------------------------------
        // (c) Update previous state
        // --------------------------------------------------------
        aPrevState[i] := aUnits[i].bPresVal;
    END_IF
END_FOR

// ------------------------------------------------------------
// Optional debug info
// ------------------------------------------------------------
sDebug := CONCAT('Queued=', INT_TO_STRING(g_iCount));

END_FUNCTION_BLOCK

// ---- POUs/FB_EventLogger/FB_EventF10.TcPOU
FUNCTION_BLOCK FB_EventF10
VAR_INPUT
	FB_Bacnet : FB_BACnet_DAIKIN_MasterStation_III_No_3;
    FB_Bacnet_b : FB_BACnet_DAIKIN_MasterStation_III_No_2;
END_VAR
VAR_OUTPUT
	sDebug : STRING(200);
END_VAR
VAR
	fbMsg : FB_TcMessage;
	aUnits : ARRAY[1..24] OF AC_Unit_Status;
	stUnit   : AC_Unit_Status;
	i: INT;
	sMsgText: STRING;
END_VAR
VAR RETAIN
	aPrevState : ARRAY[1..24] OF BOOL := [FALSE(*24*)];
END_VAR

// ============================================================
// 1) Map BACnet StartStopStatus points → aUnits
// ============================================================
aUnits[1].bPresVal := FB_Bacnet.StartStopStatus_064.bPresVal;
aUnits[1].sUnitName := 'F10-A1 (1-00)';
aUnits[2].bPresVal := FB_Bacnet.StartStopStatus_065.bPresVal;
aUnits[2].sUnitName := 'F10-A2 (1-01)';
aUnits[3].bPresVal := FB_Bacnet.StartStopStatus_066.bPresVal;
aUnits[3].sUnitName := 'F10-A3 (1-02)';
aUnits[4].bPresVal := FB_Bacnet.StartStopStatus_067.bPresVal;
aUnits[4].sUnitName := 'F10-A4 (1-03)';
aUnits[5].bPresVal := FB_Bacnet.StartStopStatus_068.bPresVal;
aUnits[5].sUnitName := 'F10-B1 (1-04)';
aUnits[6].bPresVal := FB_Bacnet.StartStopStatus_069.bPresVal;
aUnits[6].sUnitName := 'F10-B2 (1-05)';
aUnits[7].bPresVal := FB_Bacnet.StartStopStatus_070.bPresVal;
aUnits[7].sUnitName := 'F10-C1 (1-06)';
aUnits[8].bPresVal := FB_Bacnet.StartStopStatus_071.bPresVal;
aUnits[8].sUnitName := 'F10-C2 (1-07)';
aUnits[9].bPresVal := FB_Bacnet.StartStopStatus_072.bPresVal;
aUnits[9].sUnitName := 'F10-D1 (1-08)';
aUnits[10].bPresVal := FB_Bacnet.StartStopStatus_073.bPresVal;
aUnits[10].sUnitName := 'F10-D2 (1-09)';
aUnits[11].bPresVal := FB_Bacnet.StartStopStatus_074.bPresVal;
aUnits[11].sUnitName := 'F10-D3 (1-10)';
aUnits[12].bPresVal := FB_Bacnet.StartStopStatus_075.bPresVal;
aUnits[12].sUnitName := 'F10-D4 (1-11)';
aUnits[13].bPresVal := FB_Bacnet.StartStopStatus_076.bPresVal;
aUnits[13].sUnitName := 'F10-D5 (1-12)';
aUnits[14].bPresVal := FB_Bacnet.StartStopStatus_077.bPresVal;
aUnits[14].sUnitName := 'F10-D6 (1-13)';
aUnits[15].bPresVal := FB_Bacnet.StartStopStatus_078.bPresVal;
aUnits[15].sUnitName := 'F10-E1 (1-14)';
aUnits[16].bPresVal := FB_Bacnet.StartStopStatus_079.bPresVal;
aUnits[16].sUnitName := 'F10-E2 (1-15)';
aUnits[17].bPresVal := FB_Bacnet.StartStopStatus_080.bPresVal;
aUnits[17].sUnitName := 'F10-F1 (2-00)';
aUnits[18].bPresVal := FB_Bacnet.StartStopStatus_081.bPresVal;
aUnits[18].sUnitName := 'F10-F2 (2-01)';
aUnits[19].bPresVal := FB_Bacnet.StartStopStatus_082.bPresVal;
aUnits[19].sUnitName := 'F10-G1 (2-02)';
aUnits[20].bPresVal := FB_Bacnet.StartStopStatus_083.bPresVal;
aUnits[20].sUnitName := 'F10-G2 (2-03)';
aUnits[21].bPresVal := FB_Bacnet.StartStopStatus_084.bPresVal;
aUnits[21].sUnitName := 'F10-G3 (2-04)';
aUnits[22].bPresVal := FB_Bacnet.StartStopStatus_112.bPresVal;
aUnits[22].sUnitName := 'F10-IT1 (4-00)';
//aUnits[23].bPresVal := FB_Bacnet.StartStopStatus_241.bPresVal;
//aUnits[23].sUnitName := 'F10-IT2 (4-01)';
aUnits[24].bPresVal := FB_Bacnet.StartStopStatus_226.bPresVal;
aUnits[24].sUnitName := 'F10-Lobi (3-02)';

// ============================================================
// 2) Detect changes & handle events
// ============================================================

FOR i := 1 TO 24 DO
    stUnit := aUnits[i];

    // Detect ON/OFF state change
    IF aUnits[i].bPresVal <> aPrevState[i] THEN
        // --------------------------------------------------------
        // (a) Send TwinCAT message as before
        // --------------------------------------------------------
        IF aUnits[i].bPresVal THEN
            sMsgText := CONCAT(stUnit.sUnitName, ' is Turned ON');
        ELSE
            sMsgText := CONCAT(stUnit.sUnitName, ' is Turned OFF');
        END_IF

        fbMsg.CreateEx(TC_EVENTS.UnitPowerStatus.EventPowerStatus, 0);
        fbMsg.ipArguments.AddString(sMsgText);
        fbMsg.Send(0);

        // --------------------------------------------------------
        // (b) Push event to global CSV queue (for P_CSVWrite_TextMode)
        // --------------------------------------------------------
        IF g_iCount < g_CSV_BUF_SIZE THEN
            g_aUnitName[g_iWriteIdx] := stUnit.sUnitName;
            g_aState[g_iWriteIdx]    := aUnits[i].bPresVal;
            g_iWriteIdx := g_iWriteIdx + 1;
            IF g_iWriteIdx > g_CSV_BUF_SIZE THEN g_iWriteIdx := 1; END_IF
            g_iCount := g_iCount + 1;
        END_IF

        // --------------------------------------------------------
        // (c) Update previous state
        // --------------------------------------------------------
        aPrevState[i] := aUnits[i].bPresVal;
    END_IF
END_FOR

// ------------------------------------------------------------
// Optional debug info
// ------------------------------------------------------------
sDebug := CONCAT('Queued=', INT_TO_STRING(g_iCount));

END_FUNCTION_BLOCK

// ---- POUs/FB_EventLogger/FB_EventF11.TcPOU
FUNCTION_BLOCK FB_EventF11
VAR_INPUT
	FB_Bacnet : FB_BACnet_DAIKIN_MasterStation_III_No_3;
  	FB_Bacnet_b : FB_BACnet_DAIKIN_MasterStation_III_No_2;
END_VAR
VAR_OUTPUT
	sDebug : STRING(200);
END_VAR
VAR
	fbMsg : FB_TcMessage;
	aUnits : ARRAY[1..22] OF AC_Unit_Status;
	stUnit   : AC_Unit_Status;
	i: INT;
	sMsgText: STRING;
END_VAR
VAR RETAIN
	aPrevState : ARRAY[1..22] OF BOOL := [FALSE(*22*)];
END_VAR


//aUnits[1].bPresVal := FB_Bacnet.StartStopStatus_128.bPresVal;
//aUnits[1].sUnitName := 'F11-A1 (1-00)';
//aUnits[2].bPresVal := FB_Bacnet.StartStopStatus_129.bPresVal;
//aUnits[2].sUnitName := 'F11-A2 (1-01)';
//aUnits[3].bPresVal := FB_Bacnet.StartStopStatus_130.bPresVal;
//aUnits[3].sUnitName := 'F11-A3 (1-02)';
//aUnits[4].bPresVal := FB_Bacnet.StartStopStatus_131.bPresVal;
//aUnits[4].sUnitName := 'F11-A4 (1-03)';
//aUnits[5].bPresVal := FB_Bacnet.StartStopStatus_132.bPresVal;
//aUnits[5].sUnitName := 'F11-A5 (1-04)';
//aUnits[6].bPresVal := FB_Bacnet.StartStopStatus_133.bPresVal;
//aUnits[6].sUnitName := 'F11-A6 (1-05)';
//aUnits[7].bPresVal := FB_Bacnet.StartStopStatus_134.bPresVal;
//aUnits[7].sUnitName := 'F11-B1 (1-06)';
//aUnits[8].bPresVal := FB_Bacnet.StartStopStatus_135.bPresVal;
//aUnits[8].sUnitName := 'F11-B2 (1-07)';
//aUnits[9].bPresVal := FB_Bacnet.StartStopStatus_136.bPresVal;
//aUnits[9].sUnitName := 'F11-C1 (1-08)';
//aUnits[10].bPresVal := FB_Bacnet.StartStopStatus_137.bPresVal;
//aUnits[10].sUnitName := 'F11-C2 (1-09)';
//aUnits[11].bPresVal := FB_Bacnet.StartStopStatus_138.bPresVal;
//aUnits[11].sUnitName := 'F11-D1 (1-10)';
//aUnits[12].bPresVal := FB_Bacnet.StartStopStatus_139.bPresVal;
//aUnits[12].sUnitName := 'F11-D2 (1-11)';
//aUnits[13].bPresVal := FB_Bacnet.StartStopStatus_140.bPresVal;
//aUnits[13].sUnitName := 'F11-D3 (1-12)';
//aUnits[14].bPresVal := FB_Bacnet.StartStopStatus_141.bPresVal;
//aUnits[14].sUnitName := 'F11-D4 (1-13)';
//aUnits[15].bPresVal := FB_Bacnet.StartStopStatus_142.bPresVal;
//aUnits[15].sUnitName := 'F11-E1 (1-14)';
//aUnits[16].bPresVal := FB_Bacnet.StartStopStatus_143.bPresVal;
//aUnits[16].sUnitName := 'F11-E2 (1-15)';
aUnits[17].bPresVal := FB_Bacnet.StartStopStatus_144.bPresVal;
aUnits[17].sUnitName := 'F11-E3 (2-00)';
//aUnits[18].bPresVal := FB_Bacnet.StartStopStatus_145.bPresVal;
//aUnits[18].sUnitName := 'F11-F1 (2-01)';
//aUnits[19].bPresVal := FB_Bacnet.StartStopStatus_146.bPresVal;
//aUnits[19].sUnitName := 'F11-F2 (2-02)';
//aUnits[20].bPresVal := FB_Bacnet.StartStopStatus_147.bPresVal;
//aUnits[20].sUnitName := 'F11-G1 (2-03)';
//aUnits[21].bPresVal := FB_Bacnet.StartStopStatus_148.bPresVal;
//aUnits[21].sUnitName := 'F11-G2 (2-04)';
aUnits[22].bPresVal := FB_Bacnet_b.StartStopStatus_227.bPresVal;
aUnits[22].sUnitName := 'F11-Lobi (3-03)';


// ============================================================
// 2) Detect changes & handle events
// ============================================================

FOR i := 1 TO 22 DO
    stUnit := aUnits[i];

    // Detect ON/OFF state change
    IF aUnits[i].bPresVal <> aPrevState[i] THEN
        // --------------------------------------------------------
        // (a) Send TwinCAT message as before
        // --------------------------------------------------------
        IF aUnits[i].bPresVal THEN
            sMsgText := CONCAT(stUnit.sUnitName, ' is Turned ON');
        ELSE
            sMsgText := CONCAT(stUnit.sUnitName, ' is Turned OFF');
        END_IF

        fbMsg.CreateEx(TC_EVENTS.UnitPowerStatus.EventPowerStatus, 0);
        fbMsg.ipArguments.AddString(sMsgText);
        fbMsg.Send(0);

        // --------------------------------------------------------
        // (b) Push event to global CSV queue (for P_CSVWrite_TextMode)
        // --------------------------------------------------------
        IF g_iCount < g_CSV_BUF_SIZE THEN
            g_aUnitName[g_iWriteIdx] := stUnit.sUnitName;
            g_aState[g_iWriteIdx]    := aUnits[i].bPresVal;
            g_iWriteIdx := g_iWriteIdx + 1;
            IF g_iWriteIdx > g_CSV_BUF_SIZE THEN g_iWriteIdx := 1; END_IF
            g_iCount := g_iCount + 1;
        END_IF

        // --------------------------------------------------------
        // (c) Update previous state
        // --------------------------------------------------------
        aPrevState[i] := aUnits[i].bPresVal;
    END_IF
END_FOR

// ------------------------------------------------------------
// Optional debug info
// ------------------------------------------------------------
sDebug := CONCAT('Queued=', INT_TO_STRING(g_iCount));

END_FUNCTION_BLOCK

// ---- POUs/FB_EventLogger/FB_EventF12.TcPOU
FUNCTION_BLOCK FB_EventF12
VAR_INPUT
	FB_Bacnet : FB_BACnet_DAIKIN_MasterStation_III_No_3;
END_VAR
VAR_OUTPUT
	sDebug : STRING(200);
END_VAR
VAR
	fbMsg : FB_TcMessage;
	aUnits : ARRAY[1..24] OF AC_Unit_Status;
	stUnit   : AC_Unit_Status;
	i: INT;
	sMsgText: STRING;
END_VAR
VAR RETAIN
	aPrevState : ARRAY[1..24] OF BOOL := [FALSE(*24*)];
END_VAR

// ============================================================
// 1) Map BACnet StartStopStatus points → aUnits
// ============================================================
//aUnits[1].bPresVal := FB_Bacnet.StartStopStatus_192.bPresVal;
//aUnits[1].sUnitName := 'F12-A1 (1-00)';
//aUnits[2].bPresVal := FB_Bacnet.StartStopStatus_193.bPresVal;
//aUnits[2].sUnitName := 'F12-A2 (1-01)';
//aUnits[3].bPresVal := FB_Bacnet.StartStopStatus_194.bPresVal;
//aUnits[3].sUnitName := 'F12-A3 (1-02)';
//aUnits[4].bPresVal := FB_Bacnet.StartStopStatus_195.bPresVal;
//aUnits[4].sUnitName := 'F12-A4 (1-03)';
//aUnits[5].bPresVal := FB_Bacnet.StartStopStatus_196.bPresVal;
//aUnits[5].sUnitName := 'F12-A5 (1-04)';
//aUnits[6].bPresVal := FB_Bacnet.StartStopStatus_197.bPresVal;
//aUnits[6].sUnitName := 'F12-A6 (1-05)';
//aUnits[7].bPresVal := FB_Bacnet.StartStopStatus_198.bPresVal;
//aUnits[7].sUnitName := 'F12-B1 (1-06)';
//aUnits[8].bPresVal := FB_Bacnet.StartStopStatus_199.bPresVal;
//aUnits[8].sUnitName := 'F12-B2 (1-07)';
//aUnits[9].bPresVal := FB_Bacnet.StartStopStatus_200.bPresVal;
//aUnits[9].sUnitName := 'F12-C1 (1-08)';
//aUnits[10].bPresVal := FB_Bacnet.StartStopStatus_201.bPresVal;
//aUnits[10].sUnitName := 'F12-C2 (1-09)';
//aUnits[11].bPresVal := FB_Bacnet.StartStopStatus_202.bPresVal;
//aUnits[11].sUnitName := 'F12-D1 (1-10)';
//aUnits[12].bPresVal := FB_Bacnet.StartStopStatus_203.bPresVal;
//aUnits[12].sUnitName := 'F12-D2 (1-11)';
//aUnits[13].bPresVal := FB_Bacnet.StartStopStatus_204.bPresVal;
//aUnits[13].sUnitName := 'F12-D3 (1-12)';
//aUnits[14].bPresVal := FB_Bacnet.StartStopStatus_205.bPresVal;
//aUnits[14].sUnitName := 'F12-D4 (1-13)';
//aUnits[15].bPresVal := FB_Bacnet.StartStopStatus_206.bPresVal;
//aUnits[15].sUnitName := 'F12-E1 (1-14)';
//aUnits[16].bPresVal := FB_Bacnet.StartStopStatus_207.bPresVal;
//aUnits[16].sUnitName := 'F12-E2 (1-15)';
//aUnits[17].bPresVal := FB_Bacnet.StartStopStatus_208.bPresVal;
//aUnits[17].sUnitName := 'F12-E3 (2-00)';
//aUnits[18].bPresVal := FB_Bacnet.StartStopStatus_209.bPresVal;
//aUnits[18].sUnitName := 'F12-F1 (2-01)';
//aUnits[19].bPresVal := FB_Bacnet.StartStopStatus_210.bPresVal;
//aUnits[19].sUnitName := 'F12-F2 (2-02)';
//aUnits[20].bPresVal := FB_Bacnet.StartStopStatus_211.bPresVal;
//aUnits[20].sUnitName := 'F12-G1 (2-03)';
//aUnits[21].bPresVal := FB_Bacnet.StartStopStatus_212.bPresVal;
//aUnits[21].sUnitName := 'F12-G2 (2-04)';
aUnits[22].bPresVal := FB_Bacnet.StartStopStatus_224.bPresVal;
aUnits[22].sUnitName := 'F12-Lobi (3-00)';
aUnits[23].bPresVal := FB_Bacnet.StartStopStatus_225.bPresVal;
aUnits[23].sUnitName := 'F12-LMR-1 (3-01)';
aUnits[24].bPresVal := FB_Bacnet.StartStopStatus_226.bPresVal;
aUnits[24].sUnitName := 'F12-LMR-2 (3-02)';

// ============================================================
// 2) Detect changes & handle events
// ============================================================

FOR i := 1 TO 24 DO
    stUnit := aUnits[i];

    // Detect ON/OFF state change
    IF aUnits[i].bPresVal <> aPrevState[i] THEN
        // --------------------------------------------------------
        // (a) Send TwinCAT message as before
        // --------------------------------------------------------
        IF aUnits[i].bPresVal THEN
            sMsgText := CONCAT(stUnit.sUnitName, ' is Turned ON');
        ELSE
            sMsgText := CONCAT(stUnit.sUnitName, ' is Turned OFF');
        END_IF

        fbMsg.CreateEx(TC_EVENTS.UnitPowerStatus.EventPowerStatus, 0);
        fbMsg.ipArguments.AddString(sMsgText);
        fbMsg.Send(0);

        // --------------------------------------------------------
        // (b) Push event to global CSV queue (for P_CSVWrite_TextMode)
        // --------------------------------------------------------
        IF g_iCount < g_CSV_BUF_SIZE THEN
            g_aUnitName[g_iWriteIdx] := stUnit.sUnitName;
            g_aState[g_iWriteIdx]    := aUnits[i].bPresVal;
            g_iWriteIdx := g_iWriteIdx + 1;
            IF g_iWriteIdx > g_CSV_BUF_SIZE THEN g_iWriteIdx := 1; END_IF
            g_iCount := g_iCount + 1;
        END_IF

        // --------------------------------------------------------
        // (c) Update previous state
        // --------------------------------------------------------
        aPrevState[i] := aUnits[i].bPresVal;
    END_IF
END_FOR

// ------------------------------------------------------------
// Optional debug info
// ------------------------------------------------------------
sDebug := CONCAT('Queued=', INT_TO_STRING(g_iCount));

END_FUNCTION_BLOCK

// ---- POUs/FB_EventLogger/FB_EventF15.TcPOU
FUNCTION_BLOCK FB_EventF15
VAR_INPUT
	FB_Bacnet : FB_BACnet_DAIKIN_MasterStation_III_No_4;
  FB_Bacnet_b : FB_BACnet_DAIKIN_MasterStation_III_No_5;
END_VAR
VAR_OUTPUT
	sDebug : STRING(200);
END_VAR
VAR
	fbMsg : FB_TcMessage;
	aUnits : ARRAY[1..23] OF AC_Unit_Status;
	stUnit   : AC_Unit_Status;
	i: INT;
	sMsgText: STRING;
END_VAR
VAR RETAIN
	aPrevState : ARRAY[1..23] OF BOOL := [FALSE(*23*)];
END_VAR


aUnits[1].bPresVal := FB_Bacnet.StartStopStatus_000.bPresVal;
aUnits[1].sUnitName := 'F15-A1 (1-00)';
aUnits[2].bPresVal := FB_Bacnet.StartStopStatus_001.bPresVal;
aUnits[2].sUnitName := 'F15-A2 (1-01)';
aUnits[3].bPresVal := FB_Bacnet.StartStopStatus_002.bPresVal;
aUnits[3].sUnitName := 'F15-A3 (1-02)';
aUnits[4].bPresVal := FB_Bacnet.StartStopStatus_003.bPresVal;
aUnits[4].sUnitName := 'F15-A4 (1-03)';
aUnits[5].bPresVal := FB_Bacnet.StartStopStatus_004.bPresVal;
aUnits[5].sUnitName := 'F15-B1 (1-04)';
aUnits[6].bPresVal := FB_Bacnet.StartStopStatus_005.bPresVal;
aUnits[6].sUnitName := 'F15-B2 (1-05)';
aUnits[7].bPresVal := FB_Bacnet.StartStopStatus_006.bPresVal;
aUnits[7].sUnitName := 'F15-C1 (1-06)';
aUnits[8].bPresVal := FB_Bacnet.StartStopStatus_007.bPresVal;
aUnits[8].sUnitName := 'F15-C2 (1-07)';
aUnits[9].bPresVal := FB_Bacnet.StartStopStatus_008.bPresVal;
aUnits[9].sUnitName := 'F15-D1 (1-08)';
aUnits[10].bPresVal := FB_Bacnet.StartStopStatus_009.bPresVal;
aUnits[10].sUnitName := 'F15-D2 (1-09)';
aUnits[11].bPresVal := FB_Bacnet.StartStopStatus_010.bPresVal;
aUnits[11].sUnitName := 'F15-D3 (1-10)';
aUnits[12].bPresVal := FB_Bacnet.StartStopStatus_011.bPresVal;
aUnits[12].sUnitName := 'F15-D4 (1-11)';
aUnits[13].bPresVal := FB_Bacnet.StartStopStatus_012.bPresVal;
aUnits[13].sUnitName := 'F15-E1 (1-12)';
aUnits[14].bPresVal := FB_Bacnet.StartStopStatus_013.bPresVal;
aUnits[14].sUnitName := 'F15-E2 (1-13)';
aUnits[15].bPresVal := FB_Bacnet.StartStopStatus_014.bPresVal;
aUnits[15].sUnitName := 'F15-E3 (1-14)';
aUnits[16].bPresVal := FB_Bacnet.StartStopStatus_015.bPresVal;
aUnits[16].sUnitName := 'F15-F1 (1-15)';
aUnits[17].bPresVal := FB_Bacnet.StartStopStatus_016.bPresVal;
aUnits[17].sUnitName := 'F15-F2 (2-00)';
aUnits[18].bPresVal := FB_Bacnet.StartStopStatus_017.bPresVal;
aUnits[18].sUnitName := 'F15-G1 (2-01)';
aUnits[19].bPresVal := FB_Bacnet.StartStopStatus_018.bPresVal;
aUnits[19].sUnitName := 'F15-G2 (2-02)';
aUnits[20].bPresVal := FB_Bacnet.StartStopStatus_019.bPresVal;
aUnits[20].sUnitName := 'F15-H (2-03)';
aUnits[21].bPresVal := FB_Bacnet.StartStopStatus_048.bPresVal;
aUnits[21].sUnitName := 'F15-IT-1 (4-00)';
aUnits[22].bPresVal := FB_Bacnet_b.StartStopStatus_049.bPresVal;
aUnits[22].sUnitName := 'F15-IT-2 (4-01)';
aUnits[23].bPresVal := FB_Bacnet_b.StartStopStatus_032.bPresVal;
aUnits[23].sUnitName := 'F15-Lobi (3-00)';

FOR i := 1 TO 23 DO
    stUnit := aUnits[i];

    // Detect ON/OFF state change
    IF aUnits[i].bPresVal <> aPrevState[i] THEN
        // --------------------------------------------------------
        // (a) Send TwinCAT message as before
        // --------------------------------------------------------
        IF aUnits[i].bPresVal THEN
            sMsgText := CONCAT(stUnit.sUnitName, ' is Turned ON');
        ELSE
            sMsgText := CONCAT(stUnit.sUnitName, ' is Turned OFF');
        END_IF

        fbMsg.CreateEx(TC_EVENTS.UnitPowerStatus.EventPowerStatus, 0);
        fbMsg.ipArguments.AddString(sMsgText);
        fbMsg.Send(0);

        // --------------------------------------------------------
        // (b) Push event to global CSV queue (for P_CSVWrite_TextMode)
        // --------------------------------------------------------
        IF g_iCount < g_CSV_BUF_SIZE THEN
            g_aUnitName[g_iWriteIdx] := stUnit.sUnitName;
            g_aState[g_iWriteIdx]    := aUnits[i].bPresVal;
            g_iWriteIdx := g_iWriteIdx + 1;
            IF g_iWriteIdx > g_CSV_BUF_SIZE THEN g_iWriteIdx := 1; END_IF
            g_iCount := g_iCount + 1;
        END_IF

        // --------------------------------------------------------
        // (c) Update previous state
        // --------------------------------------------------------
        aPrevState[i] := aUnits[i].bPresVal;
    END_IF
END_FOR

// ------------------------------------------------------------
// Optional debug info
// ------------------------------------------------------------
sDebug := CONCAT('Queued=', INT_TO_STRING(g_iCount));

END_FUNCTION_BLOCK

// ---- POUs/FB_EventLogger/FB_EventF16.TcPOU
FUNCTION_BLOCK FB_EventF16
VAR_INPUT
	FB_Bacnet : FB_BACnet_DAIKIN_MasterStation_III_No_4;
  FB_Bacnet_b : FB_BACnet_DAIKIN_MasterStation_III_No_5;
END_VAR
VAR_OUTPUT
	sDebug : STRING(200);
END_VAR
VAR
	fbMsg : FB_TcMessage;
	aUnits : ARRAY[1..21] OF AC_Unit_Status;
	stUnit   : AC_Unit_Status;
	i: INT;
	sMsgText: STRING;
END_VAR
VAR RETAIN
	aPrevState : ARRAY[1..21] OF BOOL := [FALSE(*21*)];
END_VAR


aUnits[1].bPresVal := FB_Bacnet.StartStopStatus_064.bPresVal;
aUnits[1].sUnitName := 'F16-A1 (1-00)';
aUnits[2].bPresVal := FB_Bacnet.StartStopStatus_065.bPresVal;
aUnits[2].sUnitName := 'F16-A2 (1-01)';
aUnits[3].bPresVal := FB_Bacnet.StartStopStatus_066.bPresVal;
aUnits[3].sUnitName := 'F16-A3 (1-02)';
aUnits[4].bPresVal := FB_Bacnet.StartStopStatus_067.bPresVal;
aUnits[4].sUnitName := 'F16-A4 (1-03)';
aUnits[5].bPresVal := FB_Bacnet.StartStopStatus_068.bPresVal;
aUnits[5].sUnitName := 'F16-B1 (1-04)';
aUnits[6].bPresVal := FB_Bacnet.StartStopStatus_069.bPresVal;
aUnits[6].sUnitName := 'F16-B2 (1-05)';
aUnits[7].bPresVal := FB_Bacnet.StartStopStatus_070.bPresVal;
aUnits[7].sUnitName := 'F16-C1 (1-06)';
aUnits[8].bPresVal := FB_Bacnet.StartStopStatus_071.bPresVal;
aUnits[8].sUnitName := 'F16-C2 (1-07)';
aUnits[9].bPresVal := FB_Bacnet.StartStopStatus_072.bPresVal;
aUnits[9].sUnitName := 'F16-D1 (1-08)';
aUnits[10].bPresVal := FB_Bacnet.StartStopStatus_073.bPresVal;
aUnits[10].sUnitName := 'F16-D2 (1-09)';
aUnits[11].bPresVal := FB_Bacnet.StartStopStatus_074.bPresVal;
aUnits[11].sUnitName := 'F16-D3 (1-10)';
aUnits[12].bPresVal := FB_Bacnet.StartStopStatus_075.bPresVal;
aUnits[12].sUnitName := 'F16-D4 (1-11)';
aUnits[13].bPresVal := FB_Bacnet.StartStopStatus_076.bPresVal;
aUnits[13].sUnitName := 'F16-E1 (1-12)';
aUnits[14].bPresVal := FB_Bacnet.StartStopStatus_077.bPresVal;
aUnits[14].sUnitName := 'F16-E2 (1-13)';
aUnits[15].bPresVal := FB_Bacnet.StartStopStatus_078.bPresVal;
aUnits[15].sUnitName := 'F16-E3 (1-14)';
aUnits[16].bPresVal := FB_Bacnet.StartStopStatus_079.bPresVal;
aUnits[16].sUnitName := 'F16-F1 (1-15)';
aUnits[17].bPresVal := FB_Bacnet.StartStopStatus_080.bPresVal;
aUnits[17].sUnitName := 'F16-F2 (2-00)';
aUnits[18].bPresVal := FB_Bacnet.StartStopStatus_081.bPresVal;
aUnits[18].sUnitName := 'F16-G1 (2-01)';
aUnits[19].bPresVal := FB_Bacnet.StartStopStatus_082.bPresVal;
aUnits[19].sUnitName := 'F16-G2 (2-02)';
aUnits[20].bPresVal := FB_Bacnet.StartStopStatus_083.bPresVal;
aUnits[20].sUnitName := 'F16-H (2-03)';
aUnits[21].bPresVal := FB_Bacnet_b.StartStopStatus_033.bPresVal;
aUnits[21].sUnitName := 'F16-Lobi (3-01)';

FOR i := 1 TO 21 DO
    stUnit := aUnits[i];

    // Detect ON/OFF state change
    IF aUnits[i].bPresVal <> aPrevState[i] THEN
        // --------------------------------------------------------
        // (a) Send TwinCAT message as before
        // --------------------------------------------------------
        IF aUnits[i].bPresVal THEN
            sMsgText := CONCAT(stUnit.sUnitName, ' is Turned ON');
        ELSE
            sMsgText := CONCAT(stUnit.sUnitName, ' is Turned OFF');
        END_IF

        fbMsg.CreateEx(TC_EVENTS.UnitPowerStatus.EventPowerStatus, 0);
        fbMsg.ipArguments.AddString(sMsgText);
        fbMsg.Send(0);

        // --------------------------------------------------------
        // (b) Push event to global CSV queue (for P_CSVWrite_TextMode)
        // --------------------------------------------------------
        IF g_iCount < g_CSV_BUF_SIZE THEN
            g_aUnitName[g_iWriteIdx] := stUnit.sUnitName;
            g_aState[g_iWriteIdx]    := aUnits[i].bPresVal;
            g_iWriteIdx := g_iWriteIdx + 1;
            IF g_iWriteIdx > g_CSV_BUF_SIZE THEN g_iWriteIdx := 1; END_IF
            g_iCount := g_iCount + 1;
        END_IF

        // --------------------------------------------------------
        // (c) Update previous state
        // --------------------------------------------------------
        aPrevState[i] := aUnits[i].bPresVal;
    END_IF
END_FOR

// ------------------------------------------------------------
// Optional debug info
// ------------------------------------------------------------
sDebug := CONCAT('Queued=', INT_TO_STRING(g_iCount));

END_FUNCTION_BLOCK

// ---- POUs/FB_EventLogger/FB_EventF17.TcPOU
FUNCTION_BLOCK FB_EventF17
VAR_INPUT
	FB_Bacnet : FB_BACnet_DAIKIN_MasterStation_III_No_4;
  FB_Bacnet_b : FB_BACnet_DAIKIN_MasterStation_III_No_5;
END_VAR
VAR_OUTPUT
	sDebug : STRING(200);
END_VAR
VAR
	fbMsg : FB_TcMessage;
	aUnits : ARRAY[1..21] OF AC_Unit_Status;
	stUnit   : AC_Unit_Status;
	i: INT;
	sMsgText: STRING;
END_VAR
VAR RETAIN
	aPrevState : ARRAY[1..21] OF BOOL := [FALSE(*21*)];
END_VAR


aUnits[1].bPresVal := FB_Bacnet.StartStopStatus_128.bPresVal;
aUnits[1].sUnitName := 'F17-A1 (1-00)';
aUnits[2].bPresVal := FB_Bacnet.StartStopStatus_129.bPresVal;
aUnits[2].sUnitName := 'F17-A2 (1-01)';
aUnits[3].bPresVal := FB_Bacnet.StartStopStatus_130.bPresVal;
aUnits[3].sUnitName := 'F17-A3 (1-02)';
aUnits[4].bPresVal := FB_Bacnet.StartStopStatus_131.bPresVal;
aUnits[4].sUnitName := 'F17-A4 (1-03)';
aUnits[5].bPresVal := FB_Bacnet.StartStopStatus_132.bPresVal;
aUnits[5].sUnitName := 'F17-B1 (1-04)';
aUnits[6].bPresVal := FB_Bacnet.StartStopStatus_133.bPresVal;
aUnits[6].sUnitName := 'F17-B2 (1-05)';
aUnits[7].bPresVal := FB_Bacnet.StartStopStatus_134.bPresVal;
aUnits[7].sUnitName := 'F17-C1 (1-06)';
aUnits[8].bPresVal := FB_Bacnet.StartStopStatus_135.bPresVal;
aUnits[8].sUnitName := 'F17-C2 (1-07)';
aUnits[9].bPresVal := FB_Bacnet.StartStopStatus_136.bPresVal;
aUnits[9].sUnitName := 'F17-D1 (1-08)';
aUnits[10].bPresVal := FB_Bacnet.StartStopStatus_137.bPresVal;
aUnits[10].sUnitName := 'F17-D2 (1-09)';
aUnits[11].bPresVal := FB_Bacnet.StartStopStatus_138.bPresVal;
aUnits[11].sUnitName := 'F17-D3 (1-10)';
aUnits[12].bPresVal := FB_Bacnet.StartStopStatus_139.bPresVal;
aUnits[12].sUnitName := 'F17-D4 (1-11)';
aUnits[13].bPresVal := FB_Bacnet.StartStopStatus_140.bPresVal;
aUnits[13].sUnitName := 'F17-E1 (1-12)';
aUnits[14].bPresVal := FB_Bacnet.StartStopStatus_141.bPresVal;
aUnits[14].sUnitName := 'F17-E2 (1-13)';
aUnits[15].bPresVal := FB_Bacnet.StartStopStatus_142.bPresVal;
aUnits[15].sUnitName := 'F17-E3 (1-14)';
aUnits[16].bPresVal := FB_Bacnet.StartStopStatus_143.bPresVal;
aUnits[16].sUnitName := 'F17-F1 (1-15)';
aUnits[17].bPresVal := FB_Bacnet.StartStopStatus_144.bPresVal;
aUnits[17].sUnitName := 'F17-F2 (2-00)';
aUnits[18].bPresVal := FB_Bacnet.StartStopStatus_145.bPresVal;
aUnits[18].sUnitName := 'F17-G1 (2-01)';
aUnits[19].bPresVal := FB_Bacnet.StartStopStatus_146.bPresVal;
aUnits[19].sUnitName := 'F17-G2 (2-02)';
aUnits[20].bPresVal := FB_Bacnet.StartStopStatus_147.bPresVal;
aUnits[20].sUnitName := 'F17-H (2-03)';
aUnits[21].bPresVal := FB_Bacnet_b.StartStopStatus_034.bPresVal;
aUnits[21].sUnitName := 'F17-Lobi (3-02)';

FOR i := 1 TO 21 DO
    stUnit := aUnits[i];

    // Detect ON/OFF state change
    IF aUnits[i].bPresVal <> aPrevState[i] THEN
        // --------------------------------------------------------
        // (a) Send TwinCAT message as before
        // --------------------------------------------------------
        IF aUnits[i].bPresVal THEN
            sMsgText := CONCAT(stUnit.sUnitName, ' is Turned ON');
        ELSE
            sMsgText := CONCAT(stUnit.sUnitName, ' is Turned OFF');
        END_IF

        fbMsg.CreateEx(TC_EVENTS.UnitPowerStatus.EventPowerStatus, 0);
        fbMsg.ipArguments.AddString(sMsgText);
        fbMsg.Send(0);

        // --------------------------------------------------------
        // (b) Push event to global CSV queue (for P_CSVWrite_TextMode)
        // --------------------------------------------------------
        IF g_iCount < g_CSV_BUF_SIZE THEN
            g_aUnitName[g_iWriteIdx] := stUnit.sUnitName;
            g_aState[g_iWriteIdx]    := aUnits[i].bPresVal;
            g_iWriteIdx := g_iWriteIdx + 1;
            IF g_iWriteIdx > g_CSV_BUF_SIZE THEN g_iWriteIdx := 1; END_IF
            g_iCount := g_iCount + 1;
        END_IF

        // --------------------------------------------------------
        // (c) Update previous state
        // --------------------------------------------------------
        aPrevState[i] := aUnits[i].bPresVal;
    END_IF
END_FOR

// ------------------------------------------------------------
// Optional debug info
// ------------------------------------------------------------
sDebug := CONCAT('Queued=', INT_TO_STRING(g_iCount));

END_FUNCTION_BLOCK

// ---- POUs/FB_EventLogger/FB_EventF18.TcPOU
FUNCTION_BLOCK FB_EventF18
VAR_INPUT
	FB_Bacnet : FB_BACnet_DAIKIN_MasterStation_III_No_5;
END_VAR
VAR_OUTPUT
	sDebug : STRING(200);
END_VAR
VAR
	fbMsg : FB_TcMessage;
	aUnits : ARRAY[1..23] OF AC_Unit_Status;
	stUnit   : AC_Unit_Status;
	i: INT;
	sMsgText: STRING;

END_VAR
VAR RETAIN
	aPrevState : ARRAY[1..23] OF BOOL := [FALSE(*23*)];
END_VAR


aUnits[1].bPresVal := FB_Bacnet.StartStopStatus_000.bPresVal;
aUnits[1].sUnitName := 'F18-A1 (1-00)';
//aUnits[2].bPresVal := FB_Bacnet.StartStopStatus_001.bPresVal;
//aUnits[2].sUnitName := 'F18-A2 (1-01)';
//aUnits[3].bPresVal := FB_Bacnet.StartStopStatus_002.bPresVal;
//aUnits[3].sUnitName := 'F18-A3 (1-02)';
//aUnits[4].bPresVal := FB_Bacnet.StartStopStatus_003.bPresVal;
//aUnits[4].sUnitName := 'F18-A4 (1-03)';
//aUnits[5].bPresVal := FB_Bacnet.StartStopStatus_004.bPresVal;
//aUnits[5].sUnitName := 'F18-B1 (1-04)';
//aUnits[6].bPresVal := FB_Bacnet.StartStopStatus_005.bPresVal;
//aUnits[6].sUnitName := 'F18-B2 (1-05)';
aUnits[7].bPresVal := FB_Bacnet.StartStopStatus_006.bPresVal;
aUnits[7].sUnitName := 'F18-C1 (1-06)';
aUnits[8].bPresVal := FB_Bacnet.StartStopStatus_007.bPresVal;
aUnits[8].sUnitName := 'F18-C2 (1-07)';
aUnits[9].bPresVal := FB_Bacnet.StartStopStatus_008.bPresVal;
aUnits[9].sUnitName := 'F18-D1 (1-08)';
aUnits[10].bPresVal := FB_Bacnet.StartStopStatus_009.bPresVal;
aUnits[10].sUnitName := 'F18-D2 (1-09)';
aUnits[11].bPresVal := FB_Bacnet.StartStopStatus_010.bPresVal;
aUnits[11].sUnitName := 'F18-D3 (1-10)';
aUnits[12].bPresVal := FB_Bacnet.StartStopStatus_011.bPresVal;
aUnits[12].sUnitName := 'F18-D4 (1-11)';
aUnits[13].bPresVal := FB_Bacnet.StartStopStatus_012.bPresVal;
aUnits[13].sUnitName := 'F18-E1 (1-12)';
aUnits[14].bPresVal := FB_Bacnet.StartStopStatus_013.bPresVal;
aUnits[14].sUnitName := 'F18-E2 (1-13)';
aUnits[15].bPresVal := FB_Bacnet.StartStopStatus_014.bPresVal;
aUnits[15].sUnitName := 'F18-E3 (1-14)';
//aUnits[16].bPresVal := FB_Bacnet.StartStopStatus_015.bPresVal;
//aUnits[16].sUnitName := 'F18-F1 (1-15)';
//aUnits[17].bPresVal := FB_Bacnet.StartStopStatus_016.bPresVal;
//aUnits[17].sUnitName := 'F18-F2 (2-00)';
aUnits[18].bPresVal := FB_Bacnet.StartStopStatus_017.bPresVal;
aUnits[18].sUnitName := 'F18-G1 (2-01)';
aUnits[19].bPresVal := FB_Bacnet.StartStopStatus_018.bPresVal;
aUnits[19].sUnitName := 'F18-G2 (2-02)';
//aUnits[20].bPresVal := FB_Bacnet.StartStopStatus_019.bPresVal;
//aUnits[20].sUnitName := 'F18-H (2-03)';
aUnits[21].bPresVal := FB_Bacnet.StartStopStatus_050.bPresVal;
aUnits[21].sUnitName := 'F18-IT-1 (4-02)';
aUnits[22].bPresVal := FB_Bacnet.StartStopStatus_051.bPresVal;
aUnits[22].sUnitName := 'F18-IT-2 (4-03)';
aUnits[23].bPresVal := FB_Bacnet.StartStopStatus_035.bPresVal;
aUnits[23].sUnitName := 'F18-Lobi (3-03)';

FOR i := 1 TO 23 DO
    stUnit := aUnits[i];

    // Detect ON/OFF state change
    IF aUnits[i].bPresVal <> aPrevState[i] THEN
        // --------------------------------------------------------
        // (a) Send TwinCAT message as before
        // --------------------------------------------------------
        IF aUnits[i].bPresVal THEN
            sMsgText := CONCAT(stUnit.sUnitName, ' is Turned ON');
        ELSE
            sMsgText := CONCAT(stUnit.sUnitName, ' is Turned OFF');
        END_IF

        fbMsg.CreateEx(TC_EVENTS.UnitPowerStatus.EventPowerStatus, 0);
        fbMsg.ipArguments.AddString(sMsgText);
        fbMsg.Send(0);

        // --------------------------------------------------------
        // (b) Push event to global CSV queue (for P_CSVWrite_TextMode)
        // --------------------------------------------------------
        IF g_iCount < g_CSV_BUF_SIZE THEN
            g_aUnitName[g_iWriteIdx] := stUnit.sUnitName;
            g_aState[g_iWriteIdx]    := aUnits[i].bPresVal;
            g_iWriteIdx := g_iWriteIdx + 1;
            IF g_iWriteIdx > g_CSV_BUF_SIZE THEN g_iWriteIdx := 1; END_IF
            g_iCount := g_iCount + 1;
        END_IF

        // --------------------------------------------------------
        // (c) Update previous state
        // --------------------------------------------------------
        aPrevState[i] := aUnits[i].bPresVal;
    END_IF
END_FOR

// ------------------------------------------------------------
// Optional debug info
// ------------------------------------------------------------
sDebug := CONCAT('Queued=', INT_TO_STRING(g_iCount));

END_FUNCTION_BLOCK

// ---- POUs/FB_EventLogger/FB_EventF19.TcPOU
FUNCTION_BLOCK FB_EventF19
VAR_INPUT
	FB_Bacnet : FB_BACnet_DAIKIN_MasterStation_III_No_5;
	FB_Bacnet_b : FB_BACnet_DAIKIN_MasterStation_III_No_6;
END_VAR
VAR_OUTPUT
	sDebug : STRING(200);
END_VAR
VAR
	fbMsg : FB_TcMessage;
	aUnits : ARRAY[1..21] OF AC_Unit_Status;
	stUnit   : AC_Unit_Status;
	i: INT;
	sMsgText: STRING;

END_VAR
VAR RETAIN
	aPrevState : ARRAY[1..21] OF BOOL := [FALSE(*21*)];
END_VAR


aUnits[1].bPresVal := FB_Bacnet.StartStopStatus_064.bPresVal;
aUnits[1].sUnitName := 'F19-A1 (1-00)';
aUnits[2].bPresVal := FB_Bacnet.StartStopStatus_065.bPresVal;
aUnits[2].sUnitName := 'F19-A2 (1-01)';
aUnits[3].bPresVal := FB_Bacnet.StartStopStatus_066.bPresVal;
aUnits[3].sUnitName := 'F19-A3 (1-02)';
aUnits[4].bPresVal := FB_Bacnet.StartStopStatus_067.bPresVal;
aUnits[4].sUnitName := 'F19-A4 (1-03)';
aUnits[5].bPresVal := FB_Bacnet.StartStopStatus_068.bPresVal;
aUnits[5].sUnitName := 'F19-B1 (1-04)';
aUnits[6].bPresVal := FB_Bacnet.StartStopStatus_069.bPresVal;
aUnits[6].sUnitName := 'F19-B2 (1-05)';
aUnits[7].bPresVal := FB_Bacnet.StartStopStatus_070.bPresVal;
aUnits[7].sUnitName := 'F19-C1 (1-06)';
aUnits[8].bPresVal := FB_Bacnet.StartStopStatus_071.bPresVal;
aUnits[8].sUnitName := 'F19-C2 (1-07)';
aUnits[9].bPresVal := FB_Bacnet.StartStopStatus_072.bPresVal;
aUnits[9].sUnitName := 'F19-D1 (1-08)';
aUnits[10].bPresVal := FB_Bacnet.StartStopStatus_073.bPresVal;
aUnits[10].sUnitName := 'F19-D2 (1-09)';
aUnits[11].bPresVal := FB_Bacnet.StartStopStatus_074.bPresVal;
aUnits[11].sUnitName := 'F19-D3 (1-10)';
aUnits[12].bPresVal := FB_Bacnet.StartStopStatus_075.bPresVal;
aUnits[12].sUnitName := 'F19-D4 (1-11)';
aUnits[13].bPresVal := FB_Bacnet.StartStopStatus_076.bPresVal;
aUnits[13].sUnitName := 'F19-E1 (1-12)';
aUnits[14].bPresVal := FB_Bacnet.StartStopStatus_077.bPresVal;
aUnits[14].sUnitName := 'F19-E2 (1-13)';
aUnits[15].bPresVal := FB_Bacnet.StartStopStatus_078.bPresVal;
aUnits[15].sUnitName := 'F19-E3 (1-14)';
aUnits[16].bPresVal := FB_Bacnet.StartStopStatus_079.bPresVal;
aUnits[16].sUnitName := 'F19-F1 (1-15)';
aUnits[17].bPresVal := FB_Bacnet.StartStopStatus_080.bPresVal;
aUnits[17].sUnitName := 'F19-F2 (2-00)';
aUnits[18].bPresVal := FB_Bacnet.StartStopStatus_081.bPresVal;
aUnits[18].sUnitName := 'F19-G1 (2-01)';
aUnits[19].bPresVal := FB_Bacnet.StartStopStatus_082.bPresVal;
aUnits[19].sUnitName := 'F19-G2 (2-02)';
aUnits[20].bPresVal := FB_Bacnet.StartStopStatus_083.bPresVal;
aUnits[20].sUnitName := 'F19-H (2-03)';
aUnits[21].bPresVal := FB_Bacnet_b.StartStopStatus_032.bPresVal;
aUnits[21].sUnitName := 'F19-Lobi (3-00)';

FOR i := 1 TO 21 DO
    stUnit := aUnits[i];

    // Detect ON/OFF state change
    IF aUnits[i].bPresVal <> aPrevState[i] THEN
        // --------------------------------------------------------
        // (a) Send TwinCAT message as before
        // --------------------------------------------------------
        IF aUnits[i].bPresVal THEN
            sMsgText := CONCAT(stUnit.sUnitName, ' is Turned ON');
        ELSE
            sMsgText := CONCAT(stUnit.sUnitName, ' is Turned OFF');
        END_IF

        fbMsg.CreateEx(TC_EVENTS.UnitPowerStatus.EventPowerStatus, 0);
        fbMsg.ipArguments.AddString(sMsgText);
        fbMsg.Send(0);

        // --------------------------------------------------------
        // (b) Push event to global CSV queue (for P_CSVWrite_TextMode)
        // --------------------------------------------------------
        IF g_iCount < g_CSV_BUF_SIZE THEN
            g_aUnitName[g_iWriteIdx] := stUnit.sUnitName;
            g_aState[g_iWriteIdx]    := aUnits[i].bPresVal;
            g_iWriteIdx := g_iWriteIdx + 1;
            IF g_iWriteIdx > g_CSV_BUF_SIZE THEN g_iWriteIdx := 1; END_IF
            g_iCount := g_iCount + 1;
        END_IF

        // --------------------------------------------------------
        // (c) Update previous state
        // --------------------------------------------------------
        aPrevState[i] := aUnits[i].bPresVal;
    END_IF
END_FOR

// ------------------------------------------------------------
// Optional debug info
// ------------------------------------------------------------
sDebug := CONCAT('Queued=', INT_TO_STRING(g_iCount));

END_FUNCTION_BLOCK

// ---- POUs/FB_EventLogger/FB_EventF20.TcPOU
FUNCTION_BLOCK FB_EventF20
VAR_INPUT
	FB_Bacnet : FB_BACnet_DAIKIN_MasterStation_III_No_5;
  	FB_Bacnet_b : FB_BACnet_DAIKIN_MasterStation_III_No_6;
END_VAR
VAR_OUTPUT
	sDebug : STRING(200);
END_VAR
VAR
	fbMsg : FB_TcMessage;
	aUnits : ARRAY[1..21] OF AC_Unit_Status;
	stUnit   : AC_Unit_Status;
	i: INT;
	sMsgText: STRING;

END_VAR
VAR RETAIN
	aPrevState : ARRAY[1..21] OF BOOL := [FALSE(*21*)];
END_VAR

//aUnits[1].bPresVal := FB_Bacnet.StartStopStatus_128.bPresVal;
//aUnits[1].sUnitName := 'F20-A1 (1-00)';
aUnits[2].bPresVal := FB_Bacnet.StartStopStatus_129.bPresVal;
aUnits[2].sUnitName := 'F20-A2 (1-01)';
aUnits[3].bPresVal := FB_Bacnet.StartStopStatus_130.bPresVal;
aUnits[3].sUnitName := 'F20-A3 (1-02)';
aUnits[4].bPresVal := FB_Bacnet.StartStopStatus_131.bPresVal;
aUnits[4].sUnitName := 'F20-A4 (1-03)';
//aUnits[5].bPresVal := FB_Bacnet.StartStopStatus_132.bPresVal;
//aUnits[5].sUnitName := 'F20-B1 (1-04)';
//aUnits[6].bPresVal := FB_Bacnet.StartStopStatus_133.bPresVal;
//aUnits[6].sUnitName := 'F20-B2 (1-05)';
aUnits[7].bPresVal := FB_Bacnet.StartStopStatus_134.bPresVal;
aUnits[7].sUnitName := 'F20-C1 (1-06)';
aUnits[8].bPresVal := FB_Bacnet.StartStopStatus_135.bPresVal;
aUnits[8].sUnitName := 'F20-C2 (1-07)';
aUnits[9].bPresVal := FB_Bacnet.StartStopStatus_136.bPresVal;
aUnits[9].sUnitName := 'F20-D1 (1-08)';
aUnits[10].bPresVal := FB_Bacnet.StartStopStatus_137.bPresVal;
aUnits[10].sUnitName := 'F20-D2 (1-09)';
aUnits[11].bPresVal := FB_Bacnet.StartStopStatus_138.bPresVal;
aUnits[11].sUnitName := 'F20-D3 (1-10)';
aUnits[12].bPresVal := FB_Bacnet.StartStopStatus_139.bPresVal;
aUnits[12].sUnitName := 'F20-D4 (1-11)';
//aUnits[13].bPresVal := FB_Bacnet.StartStopStatus_140.bPresVal;
//aUnits[13].sUnitName := 'F20-E1 (1-12)';
//aUnits[14].bPresVal := FB_Bacnet.StartStopStatus_141.bPresVal;
//aUnits[14].sUnitName := 'F20-E2 (1-13)';
//aUnits[15].bPresVal := FB_Bacnet.StartStopStatus_142.bPresVal;
//aUnits[15].sUnitName := 'F20-E3 (1-14)';
aUnits[16].bPresVal := FB_Bacnet.StartStopStatus_143.bPresVal;
aUnits[16].sUnitName := 'F20-F1 (1-15)';
aUnits[17].bPresVal := FB_Bacnet.StartStopStatus_144.bPresVal;
aUnits[17].sUnitName := 'F20-F2 (2-00)';
//aUnits[18].bPresVal := FB_Bacnet.StartStopStatus_145.bPresVal;
//aUnits[18].sUnitName := 'F20-G1 (2-01)';
//aUnits[19].bPresVal := FB_Bacnet.StartStopStatus_146.bPresVal;
//aUnits[19].sUnitName := 'F20-G2 (2-02)';
aUnits[20].bPresVal := FB_Bacnet.StartStopStatus_147.bPresVal;
aUnits[20].sUnitName := 'F20-H (2-03)';
aUnits[21].bPresVal := FB_Bacnet_b.StartStopStatus_033.bPresVal;
aUnits[21].sUnitName := 'F20-Lobi (3-01)';

FOR i := 1 TO 21 DO
    stUnit := aUnits[i];

    // Detect ON/OFF state change
    IF aUnits[i].bPresVal <> aPrevState[i] THEN
        // --------------------------------------------------------
        // (a) Send TwinCAT message as before
        // --------------------------------------------------------
        IF aUnits[i].bPresVal THEN
            sMsgText := CONCAT(stUnit.sUnitName, ' is Turned ON');
        ELSE
            sMsgText := CONCAT(stUnit.sUnitName, ' is Turned OFF');
        END_IF

        fbMsg.CreateEx(TC_EVENTS.UnitPowerStatus.EventPowerStatus, 0);
        fbMsg.ipArguments.AddString(sMsgText);
        fbMsg.Send(0);

        // --------------------------------------------------------
        // (b) Push event to global CSV queue (for P_CSVWrite_TextMode)
        // --------------------------------------------------------
        IF g_iCount < g_CSV_BUF_SIZE THEN
            g_aUnitName[g_iWriteIdx] := stUnit.sUnitName;
            g_aState[g_iWriteIdx]    := aUnits[i].bPresVal;
            g_iWriteIdx := g_iWriteIdx + 1;
            IF g_iWriteIdx > g_CSV_BUF_SIZE THEN g_iWriteIdx := 1; END_IF
            g_iCount := g_iCount + 1;
        END_IF

        // --------------------------------------------------------
        // (c) Update previous state
        // --------------------------------------------------------
        aPrevState[i] := aUnits[i].bPresVal;
    END_IF
END_FOR

// ------------------------------------------------------------
// Optional debug info
// ------------------------------------------------------------
sDebug := CONCAT('Queued=', INT_TO_STRING(g_iCount));

END_FUNCTION_BLOCK

// ---- POUs/FB_EventLogger/FB_EventF21.TcPOU
FUNCTION_BLOCK FB_EventF21
VAR_INPUT
	FB_Bacnet : FB_BACnet_DAIKIN_MasterStation_III_No_5;
  FB_Bacnet_b : FB_BACnet_DAIKIN_MasterStation_III_No_6;
END_VAR
VAR_OUTPUT
	sDebug : STRING(200);
END_VAR
VAR
	fbMsg : FB_TcMessage;
	aUnits : ARRAY[1..23] OF AC_Unit_Status;
	stUnit   : AC_Unit_Status;
	i: INT;
	sMsgText: STRING;

END_VAR
VAR RETAIN
	aPrevState : ARRAY[1..23] OF BOOL := [FALSE(*23*)];
END_VAR


aUnits[1].bPresVal := FB_Bacnet.StartStopStatus_192.bPresVal;
aUnits[1].sUnitName := 'F21-A1 (1-00)';
aUnits[2].bPresVal := FB_Bacnet.StartStopStatus_193.bPresVal;
aUnits[2].sUnitName := 'F21-A2 (1-01)';
aUnits[3].bPresVal := FB_Bacnet.StartStopStatus_194.bPresVal;
aUnits[3].sUnitName := 'F21-A3 (1-02)';
aUnits[4].bPresVal := FB_Bacnet.StartStopStatus_195.bPresVal;
aUnits[4].sUnitName := 'F21-A4 (1-03)';
aUnits[5].bPresVal := FB_Bacnet.StartStopStatus_196.bPresVal;
aUnits[5].sUnitName := 'F21-B1 (1-04)';
aUnits[6].bPresVal := FB_Bacnet.StartStopStatus_197.bPresVal;
aUnits[6].sUnitName := 'F21-B2 (1-05)';
aUnits[7].bPresVal := FB_Bacnet.StartStopStatus_198.bPresVal;
aUnits[7].sUnitName := 'F21-C1 (1-06)';
aUnits[8].bPresVal := FB_Bacnet.StartStopStatus_199.bPresVal;
aUnits[8].sUnitName := 'F21-C2 (1-07)';
aUnits[9].bPresVal := FB_Bacnet.StartStopStatus_200.bPresVal;
aUnits[9].sUnitName := 'F21-D1 (1-08)';
aUnits[10].bPresVal := FB_Bacnet.StartStopStatus_201.bPresVal;
aUnits[10].sUnitName := 'F21-D2 (1-09)';
aUnits[11].bPresVal := FB_Bacnet.StartStopStatus_202.bPresVal;
aUnits[11].sUnitName := 'F21-D3 (1-10)';
aUnits[12].bPresVal := FB_Bacnet.StartStopStatus_203.bPresVal;
aUnits[12].sUnitName := 'F21-D4 (1-11)';
aUnits[13].bPresVal := FB_Bacnet.StartStopStatus_204.bPresVal;
aUnits[13].sUnitName := 'F21-E1 (1-12)';
aUnits[14].bPresVal := FB_Bacnet.StartStopStatus_205.bPresVal;
aUnits[14].sUnitName := 'F21-E2 (1-13)';
aUnits[15].bPresVal := FB_Bacnet.StartStopStatus_206.bPresVal;
aUnits[15].sUnitName := 'F21-E3 (1-14)';
aUnits[16].bPresVal := FB_Bacnet.StartStopStatus_207.bPresVal;
aUnits[16].sUnitName := 'F21-F1 (1-15)';
aUnits[17].bPresVal := FB_Bacnet.StartStopStatus_208.bPresVal;
aUnits[17].sUnitName := 'F21-F2 (2-00)';
aUnits[18].bPresVal := FB_Bacnet.StartStopStatus_209.bPresVal;
aUnits[18].sUnitName := 'F21-G1 (2-01)';
aUnits[19].bPresVal := FB_Bacnet.StartStopStatus_210.bPresVal;
aUnits[19].sUnitName := 'F21-G2 (2-02)';
aUnits[20].bPresVal := FB_Bacnet.StartStopStatus_211.bPresVal;
aUnits[20].sUnitName := 'F21-H (2-03)';
aUnits[21].bPresVal := FB_Bacnet.StartStopStatus_240.bPresVal;
aUnits[21].sUnitName := 'F21-IT-1 (4-00)';
aUnits[22].bPresVal := FB_Bacnet_b.StartStopStatus_049.bPresVal;
aUnits[22].sUnitName := 'F21-IT-2 (4-01)';
aUnits[23].bPresVal := FB_Bacnet_b.StartStopStatus_034.bPresVal;
aUnits[23].sUnitName := 'F21-Lobi (3-02)';

FOR i := 1 TO 23 DO
    stUnit := aUnits[i];

    // Detect ON/OFF state change
    IF aUnits[i].bPresVal <> aPrevState[i] THEN
        // --------------------------------------------------------
        // (a) Send TwinCAT message as before
        // --------------------------------------------------------
        IF aUnits[i].bPresVal THEN
            sMsgText := CONCAT(stUnit.sUnitName, ' is Turned ON');
        ELSE
            sMsgText := CONCAT(stUnit.sUnitName, ' is Turned OFF');
        END_IF

        fbMsg.CreateEx(TC_EVENTS.UnitPowerStatus.EventPowerStatus, 0);
        fbMsg.ipArguments.AddString(sMsgText);
        fbMsg.Send(0);

        // --------------------------------------------------------
        // (b) Push event to global CSV queue (for P_CSVWrite_TextMode)
        // --------------------------------------------------------
        IF g_iCount < g_CSV_BUF_SIZE THEN
            g_aUnitName[g_iWriteIdx] := stUnit.sUnitName;
            g_aState[g_iWriteIdx]    := aUnits[i].bPresVal;
            g_iWriteIdx := g_iWriteIdx + 1;
            IF g_iWriteIdx > g_CSV_BUF_SIZE THEN g_iWriteIdx := 1; END_IF
            g_iCount := g_iCount + 1;
        END_IF

        // --------------------------------------------------------
        // (c) Update previous state
        // --------------------------------------------------------
        aPrevState[i] := aUnits[i].bPresVal;
    END_IF
END_FOR

// ------------------------------------------------------------
// Optional debug info
// ------------------------------------------------------------
sDebug := CONCAT('Queued=', INT_TO_STRING(g_iCount));

END_FUNCTION_BLOCK

// ---- POUs/FB_EventLogger/FB_EventF22.TcPOU
FUNCTION_BLOCK FB_EventF22
VAR_INPUT
	FB_Bacnet : FB_BACnet_DAIKIN_MasterStation_III_No_6;
END_VAR
VAR_OUTPUT
	sDebug : STRING(200);
END_VAR
VAR
	fbMsg : FB_TcMessage;
	aUnits : ARRAY[1..21] OF AC_Unit_Status;
	stUnit   : AC_Unit_Status;
	i: INT;
	sMsgText: STRING;

END_VAR
VAR RETAIN
	aPrevState : ARRAY[1..21] OF BOOL := [FALSE(*21*)];
END_VAR


aUnits[1].bPresVal := FB_Bacnet.StartStopStatus_000.bPresVal;
aUnits[1].sUnitName := 'F22-A1 (1-00)';
aUnits[2].bPresVal := FB_Bacnet.StartStopStatus_001.bPresVal;
aUnits[2].sUnitName := 'F22-A2 (1-01)';
aUnits[3].bPresVal := FB_Bacnet.StartStopStatus_002.bPresVal;
aUnits[3].sUnitName := 'F22-A3 (1-02)';
aUnits[4].bPresVal := FB_Bacnet.StartStopStatus_003.bPresVal;
aUnits[4].sUnitName := 'F22-A4 (1-03)';
aUnits[5].bPresVal := FB_Bacnet.StartStopStatus_004.bPresVal;
aUnits[5].sUnitName := 'F22-B1 (1-04)';
aUnits[6].bPresVal := FB_Bacnet.StartStopStatus_005.bPresVal;
aUnits[6].sUnitName := 'F22-B2 (1-05)';
aUnits[7].bPresVal := FB_Bacnet.StartStopStatus_006.bPresVal;
aUnits[7].sUnitName := 'F22-C1 (1-06)';
aUnits[8].bPresVal := FB_Bacnet.StartStopStatus_007.bPresVal;
aUnits[8].sUnitName := 'F22-C2 (1-07)';
aUnits[9].bPresVal := FB_Bacnet.StartStopStatus_008.bPresVal;
aUnits[9].sUnitName := 'F22-D1 (1-08)';
aUnits[10].bPresVal := FB_Bacnet.StartStopStatus_009.bPresVal;
aUnits[10].sUnitName := 'F22-D2 (1-09)';
aUnits[11].bPresVal := FB_Bacnet.StartStopStatus_010.bPresVal;
aUnits[11].sUnitName := 'F22-D3 (1-10)';
aUnits[12].bPresVal := FB_Bacnet.StartStopStatus_011.bPresVal;
aUnits[12].sUnitName := 'F22-D4 (1-11)';
aUnits[13].bPresVal := FB_Bacnet.StartStopStatus_012.bPresVal;
aUnits[13].sUnitName := 'F22-E1 (1-12)';
aUnits[14].bPresVal := FB_Bacnet.StartStopStatus_013.bPresVal;
aUnits[14].sUnitName := 'F22-E2 (1-13)';
aUnits[15].bPresVal := FB_Bacnet.StartStopStatus_014.bPresVal;
aUnits[15].sUnitName := 'F22-E3 (1-14)';
aUnits[16].bPresVal := FB_Bacnet.StartStopStatus_015.bPresVal;
aUnits[16].sUnitName := 'F22-F1 (1-15)';
aUnits[17].bPresVal := FB_Bacnet.StartStopStatus_016.bPresVal;
aUnits[17].sUnitName := 'F22-F2 (2-00)';
aUnits[18].bPresVal := FB_Bacnet.StartStopStatus_017.bPresVal;
aUnits[18].sUnitName := 'F22-G1 (2-01)';
aUnits[19].bPresVal := FB_Bacnet.StartStopStatus_018.bPresVal;
aUnits[19].sUnitName := 'F22-G2 (2-02)';
aUnits[20].bPresVal := FB_Bacnet.StartStopStatus_019.bPresVal;
aUnits[20].sUnitName := 'F22-H (2-03)';
aUnits[21].bPresVal := FB_Bacnet.StartStopStatus_035.bPresVal;
aUnits[21].sUnitName := 'F22-Lobi (3-03)';

FOR i := 1 TO 21 DO
    stUnit := aUnits[i];

    // Detect ON/OFF state change
    IF aUnits[i].bPresVal <> aPrevState[i] THEN
        // --------------------------------------------------------
        // (a) Send TwinCAT message as before
        // --------------------------------------------------------
        IF aUnits[i].bPresVal THEN
            sMsgText := CONCAT(stUnit.sUnitName, ' is Turned ON');
        ELSE
            sMsgText := CONCAT(stUnit.sUnitName, ' is Turned OFF');
        END_IF

        fbMsg.CreateEx(TC_EVENTS.UnitPowerStatus.EventPowerStatus, 0);
        fbMsg.ipArguments.AddString(sMsgText);
        fbMsg.Send(0);

        // --------------------------------------------------------
        // (b) Push event to global CSV queue (for P_CSVWrite_TextMode)
        // --------------------------------------------------------
        IF g_iCount < g_CSV_BUF_SIZE THEN
            g_aUnitName[g_iWriteIdx] := stUnit.sUnitName;
            g_aState[g_iWriteIdx]    := aUnits[i].bPresVal;
            g_iWriteIdx := g_iWriteIdx + 1;
            IF g_iWriteIdx > g_CSV_BUF_SIZE THEN g_iWriteIdx := 1; END_IF
            g_iCount := g_iCount + 1;
        END_IF

        // --------------------------------------------------------
        // (c) Update previous state
        // --------------------------------------------------------
        aPrevState[i] := aUnits[i].bPresVal;
    END_IF
END_FOR

// ------------------------------------------------------------
// Optional debug info
// ------------------------------------------------------------
sDebug := CONCAT('Queued=', INT_TO_STRING(g_iCount));

END_FUNCTION_BLOCK

// ---- POUs/FB_EventLogger/FB_EventF23.TcPOU
FUNCTION_BLOCK FB_EventF23
VAR_INPUT
	FB_Bacnet : FB_BACnet_DAIKIN_MasterStation_III_No_6;
END_VAR
VAR_OUTPUT
	sDebug : STRING(200);
END_VAR
VAR
	fbMsg : FB_TcMessage;
	aUnits : ARRAY[1..21] OF AC_Unit_Status;
	stUnit   : AC_Unit_Status;
	i: INT;
	sMsgText: STRING;

END_VAR
VAR RETAIN
	aPrevState : ARRAY[1..21] OF BOOL := [FALSE(*21*)];
END_VAR


aUnits[1].bPresVal := FB_Bacnet.StartStopStatus_064.bPresVal;
aUnits[1].sUnitName := 'F23-A1 (1-00)';
aUnits[2].bPresVal := FB_Bacnet.StartStopStatus_065.bPresVal;
aUnits[2].sUnitName := 'F23-A2 (1-01)';
aUnits[3].bPresVal := FB_Bacnet.StartStopStatus_066.bPresVal;
aUnits[3].sUnitName := 'F23-A3 (1-02)';
aUnits[4].bPresVal := FB_Bacnet.StartStopStatus_067.bPresVal;
aUnits[4].sUnitName := 'F23-A4 (1-03)';
aUnits[5].bPresVal := FB_Bacnet.StartStopStatus_068.bPresVal;
aUnits[5].sUnitName := 'F23-B1 (1-04)';
aUnits[6].bPresVal := FB_Bacnet.StartStopStatus_069.bPresVal;
aUnits[6].sUnitName := 'F23-B2 (1-05)';
aUnits[7].bPresVal := FB_Bacnet.StartStopStatus_070.bPresVal;
aUnits[7].sUnitName := 'F23-C1 (1-06)';
aUnits[8].bPresVal := FB_Bacnet.StartStopStatus_071.bPresVal;
aUnits[8].sUnitName := 'F23-C2 (1-07)';
aUnits[9].bPresVal := FB_Bacnet.StartStopStatus_072.bPresVal;
aUnits[9].sUnitName := 'F23-D1 (1-08)';
aUnits[10].bPresVal := FB_Bacnet.StartStopStatus_073.bPresVal;
aUnits[10].sUnitName := 'F23-D2 (1-09)';
aUnits[11].bPresVal := FB_Bacnet.StartStopStatus_074.bPresVal;
aUnits[11].sUnitName := 'F23-D3 (1-10)';
aUnits[12].bPresVal := FB_Bacnet.StartStopStatus_075.bPresVal;
aUnits[12].sUnitName := 'F23-D4 (1-11)';
aUnits[13].bPresVal := FB_Bacnet.StartStopStatus_076.bPresVal;
aUnits[13].sUnitName := 'F23-E1 (1-12)';
aUnits[14].bPresVal := FB_Bacnet.StartStopStatus_077.bPresVal;
aUnits[14].sUnitName := 'F23-E2 (1-13)';
aUnits[15].bPresVal := FB_Bacnet.StartStopStatus_078.bPresVal;
aUnits[15].sUnitName := 'F23-E3 (1-14)';
aUnits[16].bPresVal := FB_Bacnet.StartStopStatus_079.bPresVal;
aUnits[16].sUnitName := 'F23-F1 (1-15)';
aUnits[17].bPresVal := FB_Bacnet.StartStopStatus_080.bPresVal;
aUnits[17].sUnitName := 'F23-F2 (2-00)';
aUnits[18].bPresVal := FB_Bacnet.StartStopStatus_081.bPresVal;
aUnits[18].sUnitName := 'F23-G1 (2-01)';
aUnits[19].bPresVal := FB_Bacnet.StartStopStatus_082.bPresVal;
aUnits[19].sUnitName := 'F23-G2 (2-02)';
aUnits[20].bPresVal := FB_Bacnet.StartStopStatus_083.bPresVal;
aUnits[20].sUnitName := 'F23-H (2-03)';
aUnits[21].bPresVal := FB_Bacnet.StartStopStatus_224.bPresVal;
aUnits[21].sUnitName := 'F23-Lobi (3-00)';

FOR i := 1 TO 21 DO
    stUnit := aUnits[i];

    // Detect ON/OFF state change
    IF aUnits[i].bPresVal <> aPrevState[i] THEN
        // --------------------------------------------------------
        // (a) Send TwinCAT message as before
        // --------------------------------------------------------
        IF aUnits[i].bPresVal THEN
            sMsgText := CONCAT(stUnit.sUnitName, ' is Turned ON');
        ELSE
            sMsgText := CONCAT(stUnit.sUnitName, ' is Turned OFF');
        END_IF

        fbMsg.CreateEx(TC_EVENTS.UnitPowerStatus.EventPowerStatus, 0);
        fbMsg.ipArguments.AddString(sMsgText);
        fbMsg.Send(0);

        // --------------------------------------------------------
        // (b) Push event to global CSV queue (for P_CSVWrite_TextMode)
        // --------------------------------------------------------
        IF g_iCount < g_CSV_BUF_SIZE THEN
            g_aUnitName[g_iWriteIdx] := stUnit.sUnitName;
            g_aState[g_iWriteIdx]    := aUnits[i].bPresVal;
            g_iWriteIdx := g_iWriteIdx + 1;
            IF g_iWriteIdx > g_CSV_BUF_SIZE THEN g_iWriteIdx := 1; END_IF
            g_iCount := g_iCount + 1;
        END_IF

        // --------------------------------------------------------
        // (c) Update previous state
        // --------------------------------------------------------
        aPrevState[i] := aUnits[i].bPresVal;
    END_IF
END_FOR

// ------------------------------------------------------------
// Optional debug info
// ------------------------------------------------------------
sDebug := CONCAT('Queued=', INT_TO_STRING(g_iCount));

END_FUNCTION_BLOCK

// ---- POUs/FB_EventLogger/FB_EventF25.TcPOU
FUNCTION_BLOCK FB_EventF25
VAR_INPUT
	FB_Bacnet : FB_BACnet_DAIKIN_MasterStation_III_No_6;
END_VAR
VAR_OUTPUT
	sDebug : STRING(200);
END_VAR
VAR
	fbMsg : FB_TcMessage;
	aUnits : ARRAY[1..23] OF AC_Unit_Status;
	stUnit   : AC_Unit_Status;
	i: INT;
	sMsgText: STRING;

END_VAR
VAR RETAIN
	aPrevState : ARRAY[1..23] OF BOOL := [FALSE(*23*)];
END_VAR


aUnits[1].bPresVal := FB_Bacnet.StartStopStatus_128.bPresVal;
aUnits[1].sUnitName := 'F25-A1 (1-00)';
aUnits[2].bPresVal := FB_Bacnet.StartStopStatus_129.bPresVal;
aUnits[2].sUnitName := 'F25-A2 (1-01)';
aUnits[3].bPresVal := FB_Bacnet.StartStopStatus_130.bPresVal;
aUnits[3].sUnitName := 'F25-A3 (1-02)';
aUnits[4].bPresVal := FB_Bacnet.StartStopStatus_131.bPresVal;
aUnits[4].sUnitName := 'F25-A4 (1-03)';
aUnits[5].bPresVal := FB_Bacnet.StartStopStatus_132.bPresVal;
aUnits[5].sUnitName := 'F25-B1 (1-04)';
aUnits[6].bPresVal := FB_Bacnet.StartStopStatus_133.bPresVal;
aUnits[6].sUnitName := 'F25-B2 (1-05)';
//aUnits[7].bPresVal := FB_Bacnet.StartStopStatus_134.bPresVal;
//aUnits[7].sUnitName := 'F25-C1 (1-06)';
//aUnits[8].bPresVal := FB_Bacnet.StartStopStatus_135.bPresVal;
//aUnits[8].sUnitName := 'F25-C2 (1-07)';
aUnits[9].bPresVal := FB_Bacnet.StartStopStatus_136.bPresVal;
aUnits[9].sUnitName := 'F25-D1 (1-08)';
aUnits[10].bPresVal := FB_Bacnet.StartStopStatus_137.bPresVal;
aUnits[10].sUnitName := 'F25-D2 (1-09)';
aUnits[11].bPresVal := FB_Bacnet.StartStopStatus_138.bPresVal;
aUnits[11].sUnitName := 'F25-D3 (1-10)';
aUnits[12].bPresVal := FB_Bacnet.StartStopStatus_139.bPresVal;
aUnits[12].sUnitName := 'F25-D4 (1-11)';
aUnits[13].bPresVal := FB_Bacnet.StartStopStatus_140.bPresVal;
aUnits[13].sUnitName := 'F25-E1 (1-12)';
aUnits[14].bPresVal := FB_Bacnet.StartStopStatus_141.bPresVal;
aUnits[14].sUnitName := 'F25-E2 (1-13)';
aUnits[15].bPresVal := FB_Bacnet.StartStopStatus_142.bPresVal;
aUnits[15].sUnitName := 'F25-E3 (1-14)';
aUnits[16].bPresVal := FB_Bacnet.StartStopStatus_143.bPresVal;
aUnits[16].sUnitName := 'F25-F1 (1-15)';
aUnits[17].bPresVal := FB_Bacnet.StartStopStatus_144.bPresVal;
aUnits[17].sUnitName := 'F25-F2 (2-00)';
aUnits[18].bPresVal := FB_Bacnet.StartStopStatus_145.bPresVal;
aUnits[18].sUnitName := 'F25-G1 (2-01)';
aUnits[19].bPresVal := FB_Bacnet.StartStopStatus_146.bPresVal;
aUnits[19].sUnitName := 'F25-G2 (2-02)';
aUnits[20].bPresVal := FB_Bacnet.StartStopStatus_147.bPresVal;
aUnits[20].sUnitName := 'F25-H (2-03)';
aUnits[21].bPresVal := FB_Bacnet.StartStopStatus_176.bPresVal;
aUnits[21].sUnitName := 'F25-IT-1 (4-00)';
aUnits[22].bPresVal := FB_Bacnet.StartStopStatus_241.bPresVal;
aUnits[22].sUnitName := 'F25-IT-2 (4-01)';
aUnits[23].bPresVal := FB_Bacnet.StartStopStatus_225.bPresVal;
aUnits[23].sUnitName := 'F25-Lobi (3-01)';

FOR i := 1 TO 23 DO
    stUnit := aUnits[i];

    // Detect ON/OFF state change
    IF aUnits[i].bPresVal <> aPrevState[i] THEN
        // --------------------------------------------------------
        // (a) Send TwinCAT message as before
        // --------------------------------------------------------
        IF aUnits[i].bPresVal THEN
            sMsgText := CONCAT(stUnit.sUnitName, ' is Turned ON');
        ELSE
            sMsgText := CONCAT(stUnit.sUnitName, ' is Turned OFF');
        END_IF

        fbMsg.CreateEx(TC_EVENTS.UnitPowerStatus.EventPowerStatus, 0);
        fbMsg.ipArguments.AddString(sMsgText);
        fbMsg.Send(0);

        // --------------------------------------------------------
        // (b) Push event to global CSV queue (for P_CSVWrite_TextMode)
        // --------------------------------------------------------
        IF g_iCount < g_CSV_BUF_SIZE THEN
            g_aUnitName[g_iWriteIdx] := stUnit.sUnitName;
            g_aState[g_iWriteIdx]    := aUnits[i].bPresVal;
            g_iWriteIdx := g_iWriteIdx + 1;
            IF g_iWriteIdx > g_CSV_BUF_SIZE THEN g_iWriteIdx := 1; END_IF
            g_iCount := g_iCount + 1;
        END_IF

        // --------------------------------------------------------
        // (c) Update previous state
        // --------------------------------------------------------
        aPrevState[i] := aUnits[i].bPresVal;
    END_IF
END_FOR

// ------------------------------------------------------------
// Optional debug info
// ------------------------------------------------------------
sDebug := CONCAT('Queued=', INT_TO_STRING(g_iCount));

END_FUNCTION_BLOCK

// ---- POUs/FB_EventLogger/FB_EventF26.TcPOU
FUNCTION_BLOCK FB_EventF26
VAR_INPUT
	FB_Bacnet : FB_BACnet_DAIKIN_MasterStation_III_No_6;
END_VAR
VAR_OUTPUT
	sDebug : STRING(200);
END_VAR
VAR
	fbMsg : FB_TcMessage;
	aUnits : ARRAY[1..21] OF AC_Unit_Status;
	stUnit   : AC_Unit_Status;
	i: INT;
	sMsgText: STRING;

END_VAR
VAR RETAIN
	aPrevState : ARRAY[1..21] OF BOOL := [FALSE(*21*)];
END_VAR


aUnits[1].bPresVal := FB_Bacnet.StartStopStatus_192.bPresVal;
aUnits[1].sUnitName := 'F26-A1 (1-00)';
aUnits[2].bPresVal := FB_Bacnet.StartStopStatus_193.bPresVal;
aUnits[2].sUnitName := 'F26-A2 (1-01)';
aUnits[3].bPresVal := FB_Bacnet.StartStopStatus_194.bPresVal;
aUnits[3].sUnitName := 'F26-A3 (1-02)';
aUnits[4].bPresVal := FB_Bacnet.StartStopStatus_195.bPresVal;
aUnits[4].sUnitName := 'F26-A4 (1-03)';
aUnits[5].bPresVal := FB_Bacnet.StartStopStatus_196.bPresVal;
aUnits[5].sUnitName := 'F26-B1 (1-04)';
aUnits[6].bPresVal := FB_Bacnet.StartStopStatus_197.bPresVal;
aUnits[6].sUnitName := 'F26-B2 (1-05)';
aUnits[7].bPresVal := FB_Bacnet.StartStopStatus_198.bPresVal;
aUnits[7].sUnitName := 'F26-C1 (1-06)';
aUnits[8].bPresVal := FB_Bacnet.StartStopStatus_199.bPresVal;
aUnits[8].sUnitName := 'F26-C2 (1-07)';
aUnits[9].bPresVal := FB_Bacnet.StartStopStatus_200.bPresVal;
aUnits[9].sUnitName := 'F26-D1 (1-08)';
aUnits[10].bPresVal := FB_Bacnet.StartStopStatus_201.bPresVal;
aUnits[10].sUnitName := 'F26-D2 (1-09)';
aUnits[11].bPresVal := FB_Bacnet.StartStopStatus_202.bPresVal;
aUnits[11].sUnitName := 'F26-D3 (1-10)';
aUnits[12].bPresVal := FB_Bacnet.StartStopStatus_203.bPresVal;
aUnits[12].sUnitName := 'F26-D4 (1-11)';
aUnits[13].bPresVal := FB_Bacnet.StartStopStatus_204.bPresVal;
aUnits[13].sUnitName := 'F26-E1 (1-12)';
aUnits[14].bPresVal := FB_Bacnet.StartStopStatus_205.bPresVal;
aUnits[14].sUnitName := 'F26-E2 (1-13)';
aUnits[15].bPresVal := FB_Bacnet.StartStopStatus_206.bPresVal;
aUnits[15].sUnitName := 'F26-E3 (1-14)';
aUnits[16].bPresVal := FB_Bacnet.StartStopStatus_207.bPresVal;
aUnits[16].sUnitName := 'F26-F1 (1-15)';
aUnits[17].bPresVal := FB_Bacnet.StartStopStatus_208.bPresVal;
aUnits[17].sUnitName := 'F26-F2 (2-00)';
aUnits[18].bPresVal := FB_Bacnet.StartStopStatus_209.bPresVal;
aUnits[18].sUnitName := 'F26-G1 (2-01)';
aUnits[19].bPresVal := FB_Bacnet.StartStopStatus_210.bPresVal;
aUnits[19].sUnitName := 'F26-G2 (2-02)';
aUnits[20].bPresVal := FB_Bacnet.StartStopStatus_211.bPresVal;
aUnits[20].sUnitName := 'F26-H (2-03)';
aUnits[21].bPresVal := FB_Bacnet.StartStopStatus_226.bPresVal;
aUnits[21].sUnitName := 'F26-Lobi (3-02)';

FOR i := 1 TO 21 DO
    stUnit := aUnits[i];

    // Detect ON/OFF state change
    IF aUnits[i].bPresVal <> aPrevState[i] THEN
        // --------------------------------------------------------
        // (a) Send TwinCAT message as before
        // --------------------------------------------------------
        IF aUnits[i].bPresVal THEN
            sMsgText := CONCAT(stUnit.sUnitName, ' is Turned ON');
        ELSE
            sMsgText := CONCAT(stUnit.sUnitName, ' is Turned OFF');
        END_IF

        fbMsg.CreateEx(TC_EVENTS.UnitPowerStatus.EventPowerStatus, 0);
        fbMsg.ipArguments.AddString(sMsgText);
        fbMsg.Send(0);

        // --------------------------------------------------------
        // (b) Push event to global CSV queue (for P_CSVWrite_TextMode)
        // --------------------------------------------------------
        IF g_iCount < g_CSV_BUF_SIZE THEN
            g_aUnitName[g_iWriteIdx] := stUnit.sUnitName;
            g_aState[g_iWriteIdx]    := aUnits[i].bPresVal;
            g_iWriteIdx := g_iWriteIdx + 1;
            IF g_iWriteIdx > g_CSV_BUF_SIZE THEN g_iWriteIdx := 1; END_IF
            g_iCount := g_iCount + 1;
        END_IF

        // --------------------------------------------------------
        // (c) Update previous state
        // --------------------------------------------------------
        aPrevState[i] := aUnits[i].bPresVal;
    END_IF
END_FOR

// ------------------------------------------------------------
// Optional debug info
// ------------------------------------------------------------
sDebug := CONCAT('Queued=', INT_TO_STRING(g_iCount));

END_FUNCTION_BLOCK

// ---- POUs/FB_EventLogger/FB_EventF27.TcPOU
FUNCTION_BLOCK FB_EventF27
VAR_INPUT
	FB_Bacnet : FB_BACnet_DAIKIN_MasterStation_III_No_7;
END_VAR
VAR_OUTPUT
	sDebug : STRING(200);
END_VAR
VAR
	fbMsg : FB_TcMessage;
	aUnits : ARRAY[1..21] OF AC_Unit_Status;
	stUnit   : AC_Unit_Status;
	i: INT;
	sMsgText: STRING;

END_VAR
VAR RETAIN
	aPrevState : ARRAY[1..21] OF BOOL := [FALSE(*21*)];
END_VAR


aUnits[1].bPresVal := FB_Bacnet.StartStopStatus_000.bPresVal;
aUnits[1].sUnitName := 'F27-A1 (1-00)';
aUnits[2].bPresVal := FB_Bacnet.StartStopStatus_001.bPresVal;
aUnits[2].sUnitName := 'F27-A2 (1-01)';
aUnits[3].bPresVal := FB_Bacnet.StartStopStatus_002.bPresVal;
aUnits[3].sUnitName := 'F27-A3 (1-02)';
aUnits[4].bPresVal := FB_Bacnet.StartStopStatus_003.bPresVal;
aUnits[4].sUnitName := 'F27-A4 (1-03)';
aUnits[5].bPresVal := FB_Bacnet.StartStopStatus_004.bPresVal;
aUnits[5].sUnitName := 'F27-B1 (1-04)';
aUnits[6].bPresVal := FB_Bacnet.StartStopStatus_005.bPresVal;
aUnits[6].sUnitName := 'F27-B2 (1-05)';
aUnits[7].bPresVal := FB_Bacnet.StartStopStatus_006.bPresVal;
aUnits[7].sUnitName := 'F27-C1 (1-06)';
//aUnits[8].bPresVal := FB_Bacnet.StartStopStatus_007.bPresVal;
//aUnits[8].sUnitName := 'F27-C2 (1-07)';
aUnits[9].bPresVal := FB_Bacnet.StartStopStatus_008.bPresVal;
aUnits[9].sUnitName := 'F27-D1 (1-08)';
//aUnits[10].bPresVal := FB_Bacnet.StartStopStatus_009.bPresVal;
//aUnits[10].sUnitName := 'F27-D2 (1-09)';
aUnits[11].bPresVal := FB_Bacnet.StartStopStatus_010.bPresVal;
aUnits[11].sUnitName := 'F27-D3 (1-10)';
aUnits[12].bPresVal := FB_Bacnet.StartStopStatus_011.bPresVal;
aUnits[12].sUnitName := 'F27-D4 (1-11)';
aUnits[13].bPresVal := FB_Bacnet.StartStopStatus_012.bPresVal;
aUnits[13].sUnitName := 'F27-E1 (1-12)';
aUnits[14].bPresVal := FB_Bacnet.StartStopStatus_013.bPresVal;
aUnits[14].sUnitName := 'F27-E2 (1-13)';
aUnits[15].bPresVal := FB_Bacnet.StartStopStatus_014.bPresVal;
aUnits[15].sUnitName := 'F27-E3 (1-14)';
aUnits[16].bPresVal := FB_Bacnet.StartStopStatus_015.bPresVal;
aUnits[16].sUnitName := 'F27-F1 (1-15)';
aUnits[17].bPresVal := FB_Bacnet.StartStopStatus_016.bPresVal;
aUnits[17].sUnitName := 'F27-F2 (2-00)';
aUnits[18].bPresVal := FB_Bacnet.StartStopStatus_017.bPresVal;
aUnits[18].sUnitName := 'F27-G1 (2-01)';
aUnits[19].bPresVal := FB_Bacnet.StartStopStatus_018.bPresVal;
aUnits[19].sUnitName := 'F27-G2 (2-02)';
aUnits[20].bPresVal := FB_Bacnet.StartStopStatus_019.bPresVal;
aUnits[20].sUnitName := 'F27-H (2-03)';
aUnits[21].bPresVal := FB_Bacnet.StartStopStatus_224.bPresVal;
aUnits[21].sUnitName := 'F27-Lobi (3-00)';

FOR i := 1 TO 21 DO
    stUnit := aUnits[i];

